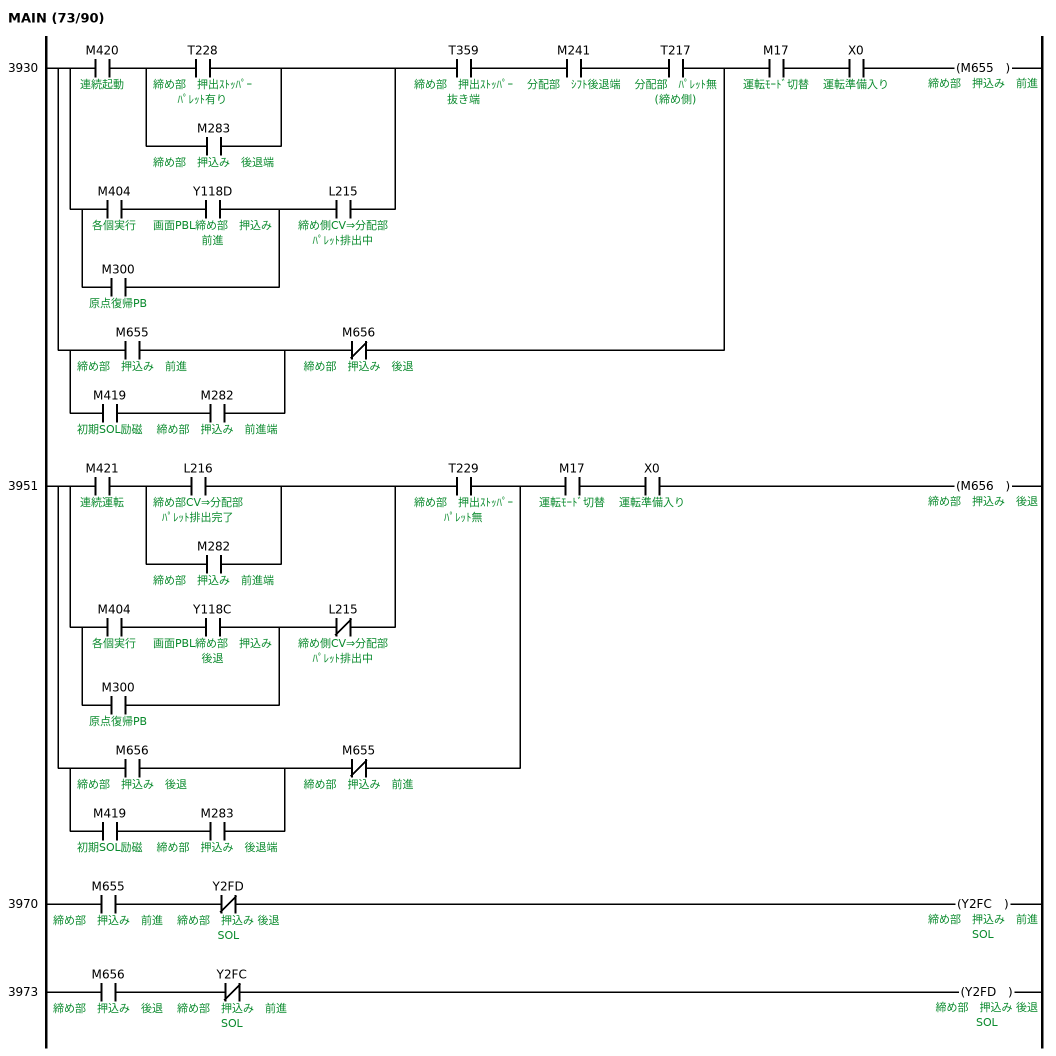
[picture p72: ladder of MAIN, rungs at steps 3930 to 3973]
3930  LD      M420  ; 連続起動
      LD      T228  ; 締め部　押出ｽﾄｯﾊﾟｰ ﾊﾟﾚｯﾄ有り
      OR      M283  ; 締め部　押込み　後退端
      ANB
      LD      M404  ; 各個実行
      AND     Y118D  ; 画面PBL締め部　押込み　前進
      OR      M300  ; 原点復帰PB
      AND     L215  ; 締め側CV⇒分配部 ﾊﾟﾚｯﾄ排出中
      ORB
      AND     T359  ; 締め部　押出ｽﾄｯﾊﾟｰ 抜き端
      AND     M241  ; 分配部　ｼﾌﾄ後退端
      AND     T217  ; 分配部　ﾊﾟﾚｯﾄ無 (締め側)
      LD      M655  ; 締め部　押込み　前進
      LD      M419  ; 初期SOL励磁
      AND     M282  ; 締め部　押込み　前進端
      ORB
      ANI     M656  ; 締め部　押込み　後退
      ORB
      AND     M17  ; 運転ﾓｰﾄﾞ切替
      AND     X0  ; 運転準備入り
      OUT     M655  ; 締め部　押込み　前進
3951  LD      M421  ; 連続運転
      LD      L216  ; 締め部CV⇒分配部 ﾊﾟﾚｯﾄ排出完了
      OR      M282  ; 締め部　押込み　前進端
      ANB
      LD      M404  ; 各個実行
      AND     Y118C  ; 画面PBL締め部　押込み　後退
      OR      M300  ; 原点復帰PB
      ANI     L215  ; 締め側CV⇒分配部 ﾊﾟﾚｯﾄ排出中
      ORB
      AND     T229  ; 締め部　押出ｽﾄｯﾊﾟｰ ﾊﾟﾚｯﾄ無
      LD      M656  ; 締め部　押込み　後退
      LD      M419  ; 初期SOL励磁
      AND     M283  ; 締め部　押込み　後退端
      ORB
      ANI     M655  ; 締め部　押込み　前進
      ORB
      AND     M17  ; 運転ﾓｰﾄﾞ切替
      AND     X0  ; 運転準備入り
      OUT     M656  ; 締め部　押込み　後退
3970  LD      M655  ; 締め部　押込み　前進
      ANI     Y2FD  ; 締め部　押込み 後退 SOL
      OUT     Y2FC  ; 締め部　押込み　前進 SOL
3973  LD      M656  ; 締め部　押込み　後退
      ANI     Y2FC  ; 締め部　押込み　前進 SOL
      OUT     Y2FD  ; 締め部　押込み 後退 SOL
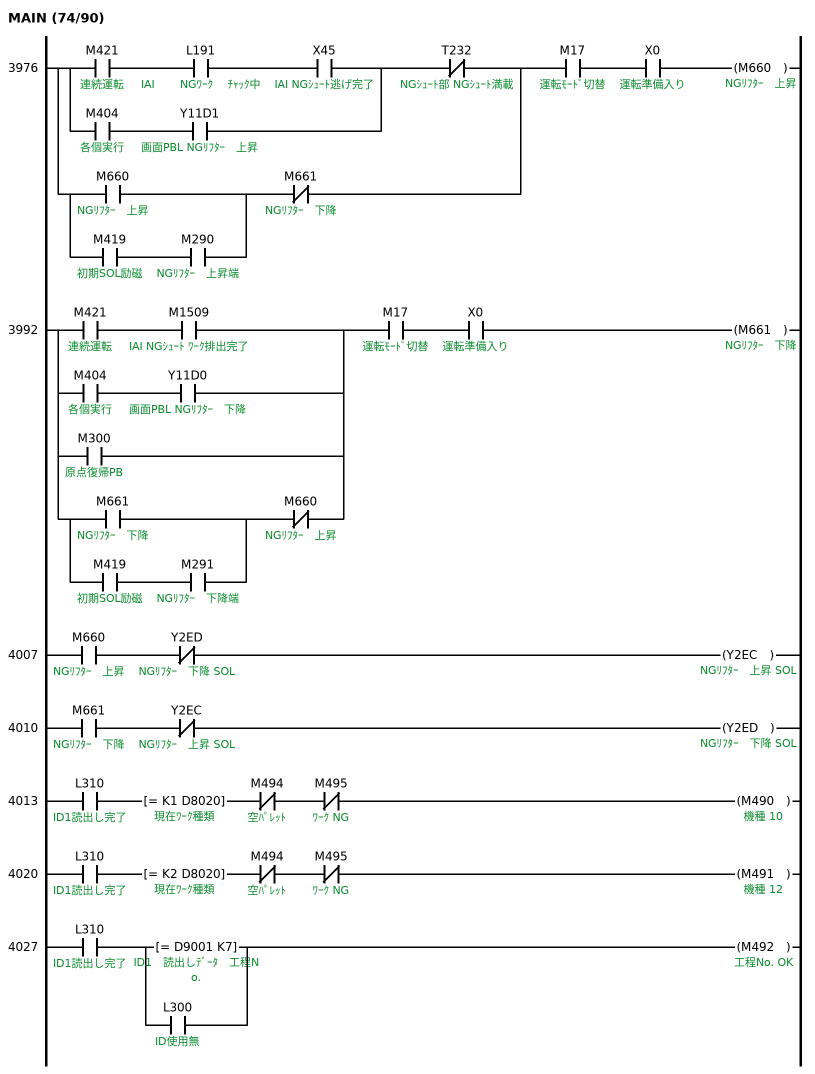
3976  LD      M421  ; 連続運転
      AND     L191  ; IAI　　 NGﾜｰｸ　 ﾁｬｯｸ中
      AND     X45  ; IAI NGｼｭｰﾄ逃げ完了
      LD      M404  ; 各個実行
      AND     Y11D1  ; 画面PBL NGﾘﾌﾀｰ　上昇
      ORB
      ANI     T232  ; NGｼｭｰﾄ部 NGｼｭｰﾄ満載
      LD      M660  ; NGﾘﾌﾀｰ　上昇
      LD      M419  ; 初期SOL励磁
      AND     M290  ; NGﾘﾌﾀｰ　上昇端
      ORB
      ANI     M661  ; NGﾘﾌﾀｰ　下降
      ORB
      AND     M17  ; 運転ﾓｰﾄﾞ切替
      AND     X0  ; 運転準備入り
      OUT     M660  ; NGﾘﾌﾀｰ　上昇
3992  LD      M421  ; 連続運転
      AND     M1509  ; IAI NGｼｭｰﾄ ﾜｰｸ排出完了
      LD      M404  ; 各個実行
      AND     Y11D0  ; 画面PBL NGﾘﾌﾀｰ　下降
      ORB
      OR      M300  ; 原点復帰PB
      LD      M661  ; NGﾘﾌﾀｰ　下降
      LD      M419  ; 初期SOL励磁
      AND     M291  ; NGﾘﾌﾀｰ　下降端
      ORB
      ANI     M660  ; NGﾘﾌﾀｰ　上昇
      ORB
      AND     M17  ; 運転ﾓｰﾄﾞ切替
      AND     X0  ; 運転準備入り
      OUT     M661  ; NGﾘﾌﾀｰ　下降
4007  LD      M660  ; NGﾘﾌﾀｰ　上昇
      ANI     Y2ED  ; NGﾘﾌﾀｰ　下降 SOL
      OUT     Y2EC  ; NGﾘﾌﾀｰ　上昇 SOL
4010  LD      M661  ; NGﾘﾌﾀｰ　下降
      ANI     Y2EC  ; NGﾘﾌﾀｰ　上昇 SOL
      OUT     Y2ED  ; NGﾘﾌﾀｰ　下降 SOL
4013  LD      L310  ; ID1読出し完了
      AND=    K1 D8020  ; 現在ﾜｰｸ種類
      ANI     M494  ; 空ﾊﾟﾚｯﾄ
      ANI     M495  ; ﾜｰｸ NG
      OUT     M490  ; 機種 10
4020  LD      L310  ; ID1読出し完了
      AND=    K2 D8020  ; 現在ﾜｰｸ種類
      ANI     M494  ; 空ﾊﾟﾚｯﾄ
      ANI     M495  ; ﾜｰｸ NG
      OUT     M491  ; 機種 12
4027  LD      L310  ; ID1読出し完了
      LD=     D9001 K7  ; ID1　読出しﾃﾞｰﾀ　工程No.
      OR      L300  ; ID使用無
      ANB
      OUT     M492  ; 工程No. OK
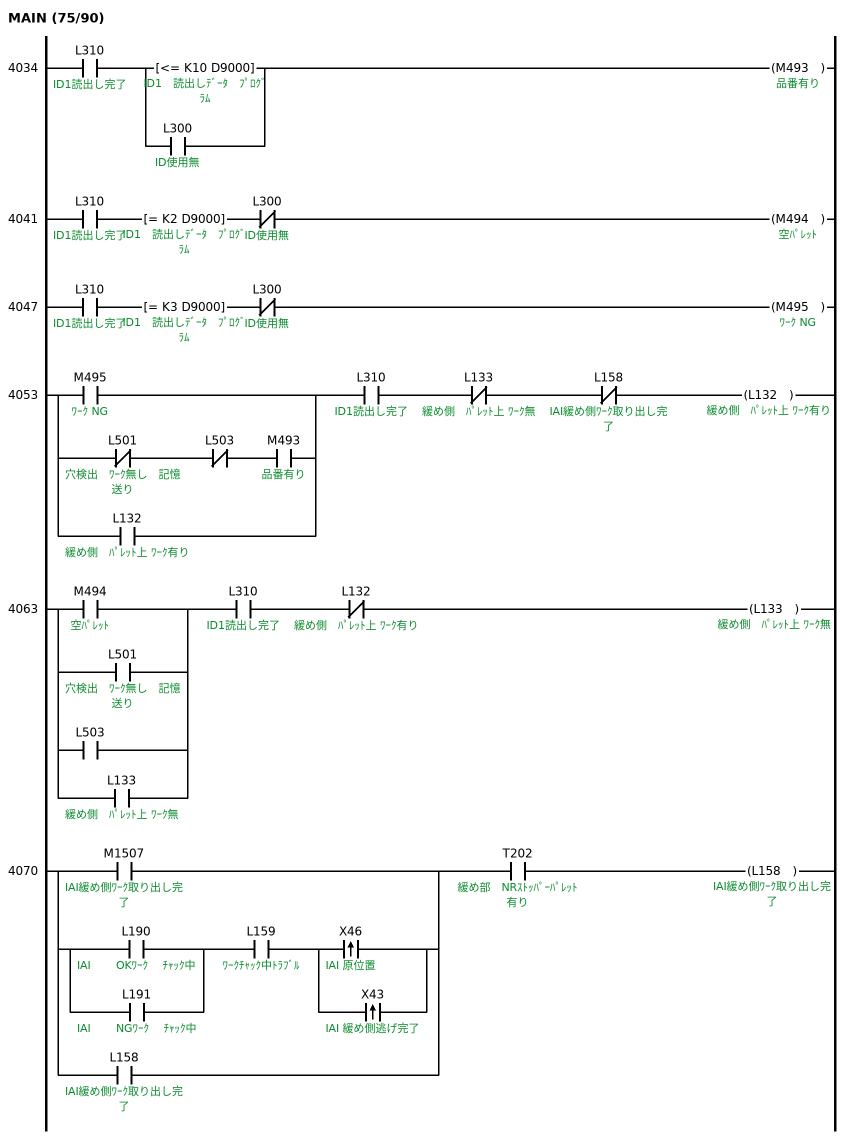
4034  LD      L310  ; ID1読出し完了
      LD<=    K10 D9000  ; ID1　読出しﾃﾞｰﾀ　ﾌﾟﾛｸﾞﾗﾑ
      OR      L300  ; ID使用無
      ANB
      OUT     M493  ; 品番有り
4041  LD      L310  ; ID1読出し完了
      AND=    K2 D9000  ; ID1　読出しﾃﾞｰﾀ　ﾌﾟﾛｸﾞﾗﾑ
      ANI     L300  ; ID使用無
      OUT     M494  ; 空ﾊﾟﾚｯﾄ
4047  LD      L310  ; ID1読出し完了
      AND=    K3 D9000  ; ID1　読出しﾃﾞｰﾀ　ﾌﾟﾛｸﾞﾗﾑ
      ANI     L300  ; ID使用無
      OUT     M495  ; ﾜｰｸ NG
4053  LD      M495  ; ﾜｰｸ NG
      LDI     L501  ; 穴検出　ﾜｰｸ無し　記憶送り
      ANI     L503
      AND     M493  ; 品番有り
      ORB
      OR      L132  ; 緩め側　ﾊﾟﾚｯﾄ上 ﾜｰｸ有り
      AND     L310  ; ID1読出し完了
      ANI     L133  ; 緩め側　ﾊﾟﾚｯﾄ上 ﾜｰｸ無
      ANI     L158  ; IAI緩め側ﾜｰｸ取り出し完了
      OUT     L132  ; 緩め側　ﾊﾟﾚｯﾄ上 ﾜｰｸ有り
4063  LD      M494  ; 空ﾊﾟﾚｯﾄ
      OR      L501  ; 穴検出　ﾜｰｸ無し　記憶送り
      OR      L503
      OR      L133  ; 緩め側　ﾊﾟﾚｯﾄ上 ﾜｰｸ無
      AND     L310  ; ID1読出し完了
      ANI     L132  ; 緩め側　ﾊﾟﾚｯﾄ上 ﾜｰｸ有り
      OUT     L133  ; 緩め側　ﾊﾟﾚｯﾄ上 ﾜｰｸ無
4070  LD      M1507  ; IAI緩め側ﾜｰｸ取り出し完了
      LD      L190  ; IAI　　 OKﾜｰｸ　 ﾁｬｯｸ中
      OR      L191  ; IAI　　 NGﾜｰｸ　 ﾁｬｯｸ中
      AND     L159  ; ﾜｰｸﾁｬｯｸ中ﾄﾗﾌﾞﾙ
      LDP     X46  ; IAI 原位置
      ORP     X43  ; IAI 緩め側逃げ完了
      ANB
      ORB
      OR      L158  ; IAI緩め側ﾜｰｸ取り出し完了
      AND     T202  ; 緩め部　NRｽﾄｯﾊﾟｰﾊﾟﾚｯﾄ有り
      OUT     L158  ; IAI緩め側ﾜｰｸ取り出し完了
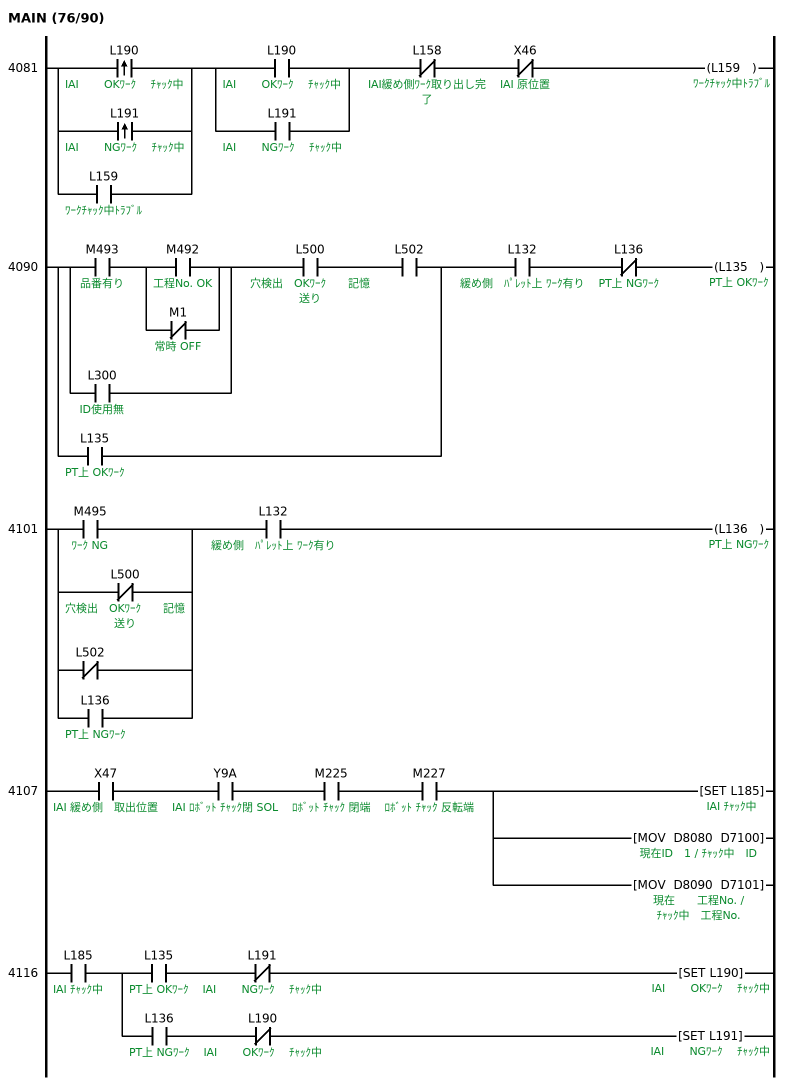
4081  LDP     L190  ; IAI　　 OKﾜｰｸ　 ﾁｬｯｸ中
      ORP     L191  ; IAI　　 NGﾜｰｸ　 ﾁｬｯｸ中
      OR      L159  ; ﾜｰｸﾁｬｯｸ中ﾄﾗﾌﾞﾙ
      LD      L190  ; IAI　　 OKﾜｰｸ　 ﾁｬｯｸ中
      OR      L191  ; IAI　　 NGﾜｰｸ　 ﾁｬｯｸ中
      ANB
      ANI     L158  ; IAI緩め側ﾜｰｸ取り出し完了
      ANI     X46  ; IAI 原位置
      OUT     L159  ; ﾜｰｸﾁｬｯｸ中ﾄﾗﾌﾞﾙ
4090  LD      M493  ; 品番有り
      LD      M492  ; 工程No. OK
      ORI     M1  ; 常時 OFF
      ANB
      OR      L300  ; ID使用無
      AND     L500  ; 穴検出　OKﾜｰｸ　　記憶送り
      AND     L502
      OR      L135  ; PT上 OKﾜｰｸ
      AND     L132  ; 緩め側　ﾊﾟﾚｯﾄ上 ﾜｰｸ有り
      ANI     L136  ; PT上 NGﾜｰｸ
      OUT     L135  ; PT上 OKﾜｰｸ
4101  LD      M495  ; ﾜｰｸ NG
      ORI     L500  ; 穴検出　OKﾜｰｸ　　記憶送り
      ORI     L502
      OR      L136  ; PT上 NGﾜｰｸ
      AND     L132  ; 緩め側　ﾊﾟﾚｯﾄ上 ﾜｰｸ有り
      OUT     L136  ; PT上 NGﾜｰｸ
4107  LD      X47  ; IAI 緩め側　取出位置
      AND     Y9A  ; IAI ﾛﾎﾞｯﾄ ﾁｬｯｸ閉 SOL
      AND     M225  ; ﾛﾎﾞｯﾄ ﾁｬｯｸ 閉端
      AND     M227  ; ﾛﾎﾞｯﾄ ﾁｬｯｸ 反転端
      SET     L185  ; IAI ﾁｬｯｸ中
      MOV     D8080 D7100  ; 現在ID　1 / ﾁｬｯｸ中　ID
      MOV     D8090 D7101  ; 現在　　工程No. / ﾁｬｯｸ中　工程No.
4116  LD      L185  ; IAI ﾁｬｯｸ中
      MPS
      AND     L135  ; PT上 OKﾜｰｸ
      ANI     L191  ; IAI　　 NGﾜｰｸ　 ﾁｬｯｸ中
      SET     L190  ; IAI　　 OKﾜｰｸ　 ﾁｬｯｸ中
      MPP
      AND     L136  ; PT上 NGﾜｰｸ
      ANI     L190  ; IAI　　 OKﾜｰｸ　 ﾁｬｯｸ中
      SET     L191  ; IAI　　 NGﾜｰｸ　 ﾁｬｯｸ中
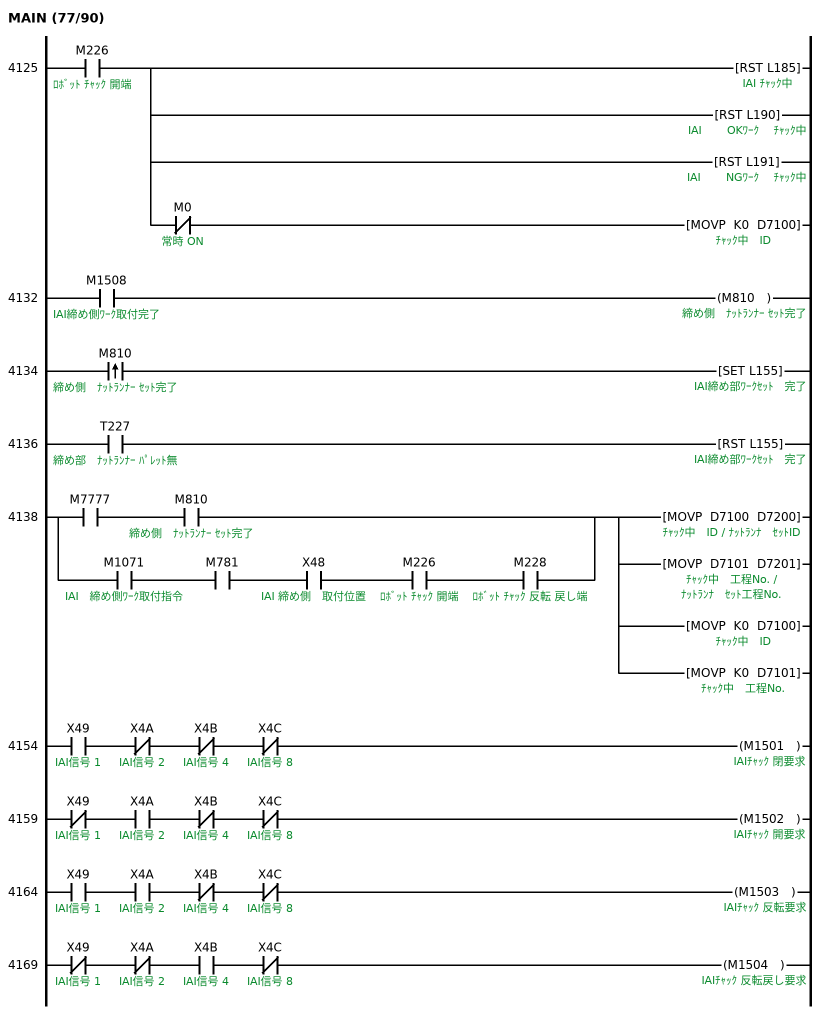
4125  LD      M226  ; ﾛﾎﾞｯﾄ ﾁｬｯｸ 開端
      RST     L185  ; IAI ﾁｬｯｸ中
      RST     L190  ; IAI　　 OKﾜｰｸ　 ﾁｬｯｸ中
      RST     L191  ; IAI　　 NGﾜｰｸ　 ﾁｬｯｸ中
      ANI     M0  ; 常時 ON
      MOVP    K0 D7100
4132  LD      M1508  ; IAI締め側ﾜｰｸ取付完了
      OUT     M810  ; 締め側　ﾅｯﾄﾗﾝﾅｰ ｾｯﾄ完了
4134  LDP     M810  ; 締め側　ﾅｯﾄﾗﾝﾅｰ ｾｯﾄ完了
      SET     L155  ; IAI締め部ﾜｰｸｾｯﾄ　完了
4136  LD      T227  ; 締め部　ﾅｯﾄﾗﾝﾅｰ ﾊﾟﾚｯﾄ無
      RST     L155  ; IAI締め部ﾜｰｸｾｯﾄ　完了
4138  LD      M7777
      AND     M810  ; 締め側　ﾅｯﾄﾗﾝﾅｰ ｾｯﾄ完了
      LD      M1071  ; IAI　締め側ﾜｰｸ取付指令
      AND     M781
      AND     X48  ; IAI 締め側　取付位置
      AND     M226  ; ﾛﾎﾞｯﾄ ﾁｬｯｸ 開端
      AND     M228  ; ﾛﾎﾞｯﾄ ﾁｬｯｸ 反転 戻し端
      ORB
      MOVP    D7100 D7200  ; ﾅｯﾄﾗﾝﾅ　ｾｯﾄID
      MOVP    D7101 D7201  ; ﾅｯﾄﾗﾝﾅ　ｾｯﾄ工程No.
      MOVP    K0 D7100
      MOVP    K0 D7101
4154  LD      X49  ; IAI信号 1
      ANI     X4A  ; IAI信号 2
      ANI     X4B  ; IAI信号 4
      ANI     X4C  ; IAI信号 8
      OUT     M1501  ; IAIﾁｬｯｸ 閉要求
4159  LDI     X49  ; IAI信号 1
      AND     X4A  ; IAI信号 2
      ANI     X4B  ; IAI信号 4
      ANI     X4C  ; IAI信号 8
      OUT     M1502  ; IAIﾁｬｯｸ 開要求
4164  LD      X49  ; IAI信号 1
      AND     X4A  ; IAI信号 2
      ANI     X4B  ; IAI信号 4
      ANI     X4C  ; IAI信号 8
      OUT     M1503  ; IAIﾁｬｯｸ 反転要求
4169  LDI     X49  ; IAI信号 1
      ANI     X4A  ; IAI信号 2
      AND     X4B  ; IAI信号 4
      ANI     X4C  ; IAI信号 8
      OUT     M1504  ; IAIﾁｬｯｸ 反転戻し要求
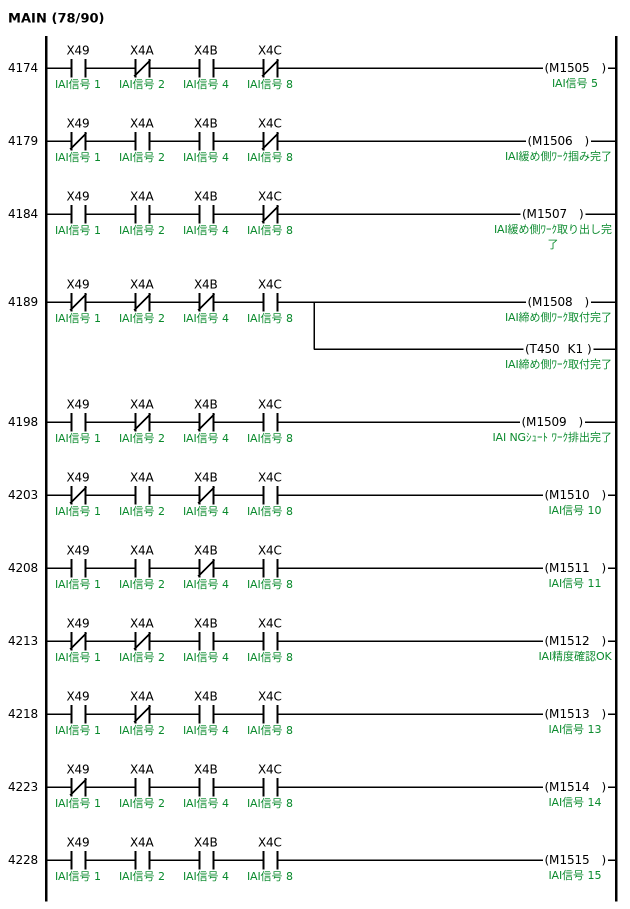
4174  LD      X49  ; IAI信号 1
      ANI     X4A  ; IAI信号 2
      AND     X4B  ; IAI信号 4
      ANI     X4C  ; IAI信号 8
      OUT     M1505  ; IAI信号 5
4179  LDI     X49  ; IAI信号 1
      AND     X4A  ; IAI信号 2
      AND     X4B  ; IAI信号 4
      ANI     X4C  ; IAI信号 8
      OUT     M1506  ; IAI緩め側ﾜｰｸ掴み完了
4184  LD      X49  ; IAI信号 1
      AND     X4A  ; IAI信号 2
      AND     X4B  ; IAI信号 4
      ANI     X4C  ; IAI信号 8
      OUT     M1507  ; IAI緩め側ﾜｰｸ取り出し完了
4189  LDI     X49  ; IAI信号 1
      ANI     X4A  ; IAI信号 2
      ANI     X4B  ; IAI信号 4
      AND     X4C  ; IAI信号 8
      OUT     M1508  ; IAI締め側ﾜｰｸ取付完了
      OUT     T450 K1  ; IAI締め側ﾜｰｸ取付完了
4198  LD      X49  ; IAI信号 1
      ANI     X4A  ; IAI信号 2
      ANI     X4B  ; IAI信号 4
      AND     X4C  ; IAI信号 8
      OUT     M1509  ; IAI NGｼｭｰﾄ ﾜｰｸ排出完了
4203  LDI     X49  ; IAI信号 1
      AND     X4A  ; IAI信号 2
      ANI     X4B  ; IAI信号 4
      AND     X4C  ; IAI信号 8
      OUT     M1510  ; IAI信号 10
4208  LD      X49  ; IAI信号 1
      AND     X4A  ; IAI信号 2
      ANI     X4B  ; IAI信号 4
      AND     X4C  ; IAI信号 8
      OUT     M1511  ; IAI信号 11
4213  LDI     X49  ; IAI信号 1
      ANI     X4A  ; IAI信号 2
      AND     X4B  ; IAI信号 4
      AND     X4C  ; IAI信号 8
      OUT     M1512  ; IAI精度確認OK
4218  LD      X49  ; IAI信号 1
      ANI     X4A  ; IAI信号 2
      AND     X4B  ; IAI信号 4
      AND     X4C  ; IAI信号 8
      OUT     M1513  ; IAI信号 13
4223  LDI     X49  ; IAI信号 1
      AND     X4A  ; IAI信号 2
      AND     X4B  ; IAI信号 4
      AND     X4C  ; IAI信号 8
      OUT     M1514  ; IAI信号 14
4228  LD      X49  ; IAI信号 1
      AND     X4A  ; IAI信号 2
      AND     X4B  ; IAI信号 4
      AND     X4C  ; IAI信号 8
      OUT     M1515  ; IAI信号 15
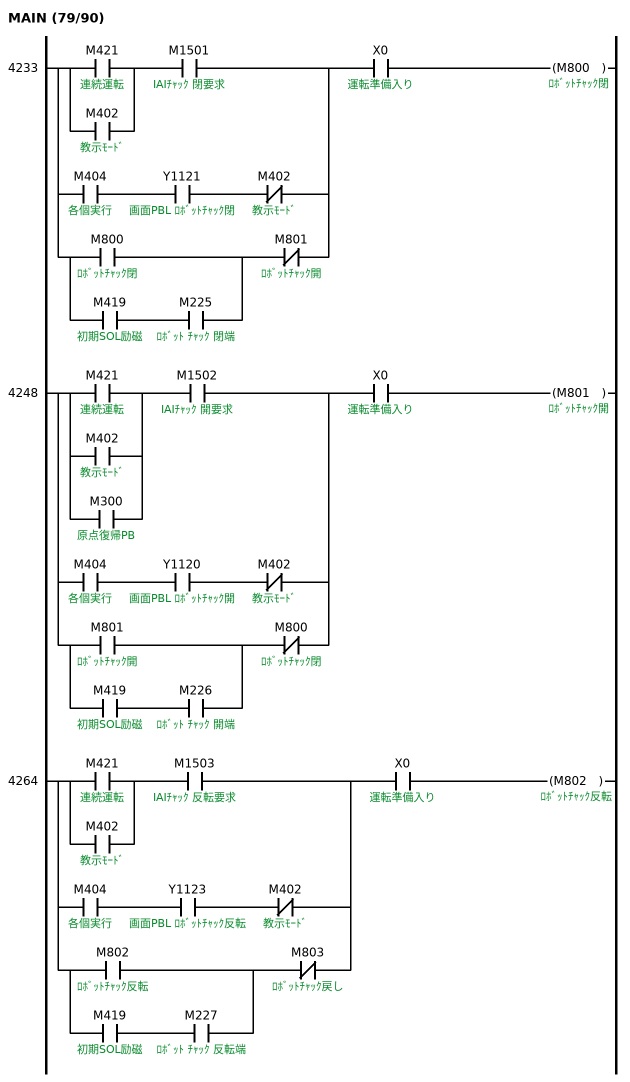
4233  LD      M421  ; 連続運転
      OR      M402  ; 教示ﾓｰﾄﾞ
      AND     M1501  ; IAIﾁｬｯｸ 閉要求
      LD      M404  ; 各個実行
      AND     Y1121  ; 画面PBL ﾛﾎﾞｯﾄﾁｬｯｸ閉
      ANI     M402  ; 教示ﾓｰﾄﾞ
      ORB
      LD      M800  ; ﾛﾎﾞｯﾄﾁｬｯｸ閉
      LD      M419  ; 初期SOL励磁
      AND     M225  ; ﾛﾎﾞｯﾄ ﾁｬｯｸ 閉端
      ORB
      ANI     M801  ; ﾛﾎﾞｯﾄﾁｬｯｸ開
      ORB
      AND     X0  ; 運転準備入り
      OUT     M800  ; ﾛﾎﾞｯﾄﾁｬｯｸ閉
4248  LD      M421  ; 連続運転
      OR      M402  ; 教示ﾓｰﾄﾞ
      OR      M300  ; 原点復帰PB
      AND     M1502  ; IAIﾁｬｯｸ 開要求
      LD      M404  ; 各個実行
      AND     Y1120  ; 画面PBL ﾛﾎﾞｯﾄﾁｬｯｸ開
      ANI     M402  ; 教示ﾓｰﾄﾞ
      ORB
      LD      M801  ; ﾛﾎﾞｯﾄﾁｬｯｸ開
      LD      M419  ; 初期SOL励磁
      AND     M226  ; ﾛﾎﾞｯﾄ ﾁｬｯｸ 開端
      ORB
      ANI     M800  ; ﾛﾎﾞｯﾄﾁｬｯｸ閉
      ORB
      AND     X0  ; 運転準備入り
      OUT     M801  ; ﾛﾎﾞｯﾄﾁｬｯｸ開
4264  LD      M421  ; 連続運転
      OR      M402  ; 教示ﾓｰﾄﾞ
      AND     M1503  ; IAIﾁｬｯｸ 反転要求
      LD      M404  ; 各個実行
      AND     Y1123  ; 画面PBL ﾛﾎﾞｯﾄﾁｬｯｸ反転
      ANI     M402  ; 教示ﾓｰﾄﾞ
      ORB
      LD      M802  ; ﾛﾎﾞｯﾄﾁｬｯｸ反転
      LD      M419  ; 初期SOL励磁
      AND     M227  ; ﾛﾎﾞｯﾄ ﾁｬｯｸ 反転端
      ORB
      ANI     M803  ; ﾛﾎﾞｯﾄﾁｬｯｸ戻し
      ORB
      AND     X0  ; 運転準備入り
      OUT     M802  ; ﾛﾎﾞｯﾄﾁｬｯｸ反転
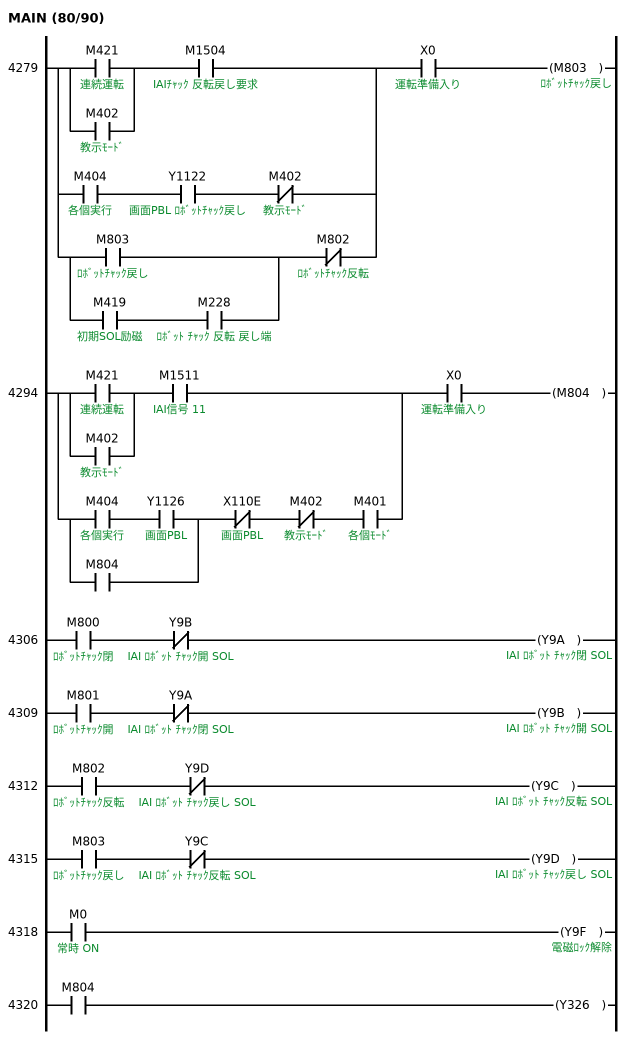
4279  LD      M421  ; 連続運転
      OR      M402  ; 教示ﾓｰﾄﾞ
      AND     M1504  ; IAIﾁｬｯｸ 反転戻し要求
      LD      M404  ; 各個実行
      AND     Y1122  ; 画面PBL ﾛﾎﾞｯﾄﾁｬｯｸ戻し
      ANI     M402  ; 教示ﾓｰﾄﾞ
      ORB
      LD      M803  ; ﾛﾎﾞｯﾄﾁｬｯｸ戻し
      LD      M419  ; 初期SOL励磁
      AND     M228  ; ﾛﾎﾞｯﾄ ﾁｬｯｸ 反転 戻し端
      ORB
      ANI     M802  ; ﾛﾎﾞｯﾄﾁｬｯｸ反転
      ORB
      AND     X0  ; 運転準備入り
      OUT     M803  ; ﾛﾎﾞｯﾄﾁｬｯｸ戻し
4294  LD      M421  ; 連続運転
      OR      M402  ; 教示ﾓｰﾄﾞ
      AND     M1511  ; IAI信号 11
      LD      M404  ; 各個実行
      AND     Y1126  ; 画面PBL
      OR      M804
      ANI     X110E  ; 画面PBL
      ANI     M402  ; 教示ﾓｰﾄﾞ
      AND     M401  ; 各個ﾓｰﾄﾞ
      ORB
      AND     X0  ; 運転準備入り
      OUT     M804
4306  LD      M800  ; ﾛﾎﾞｯﾄﾁｬｯｸ閉
      ANI     Y9B  ; IAI ﾛﾎﾞｯﾄ ﾁｬｯｸ開 SOL
      OUT     Y9A  ; IAI ﾛﾎﾞｯﾄ ﾁｬｯｸ閉 SOL
4309  LD      M801  ; ﾛﾎﾞｯﾄﾁｬｯｸ開
      ANI     Y9A  ; IAI ﾛﾎﾞｯﾄ ﾁｬｯｸ閉 SOL
      OUT     Y9B  ; IAI ﾛﾎﾞｯﾄ ﾁｬｯｸ開 SOL
4312  LD      M802  ; ﾛﾎﾞｯﾄﾁｬｯｸ反転
      ANI     Y9D  ; IAI ﾛﾎﾞｯﾄ ﾁｬｯｸ戻し SOL
      OUT     Y9C  ; IAI ﾛﾎﾞｯﾄ ﾁｬｯｸ反転 SOL
4315  LD      M803  ; ﾛﾎﾞｯﾄﾁｬｯｸ戻し
      ANI     Y9C  ; IAI ﾛﾎﾞｯﾄ ﾁｬｯｸ反転 SOL
      OUT     Y9D  ; IAI ﾛﾎﾞｯﾄ ﾁｬｯｸ戻し SOL
4318  LD      M0  ; 常時 ON
      OUT     Y9F  ; 電磁ﾛｯｸ解除
4320  LD      M804
      OUT     Y326
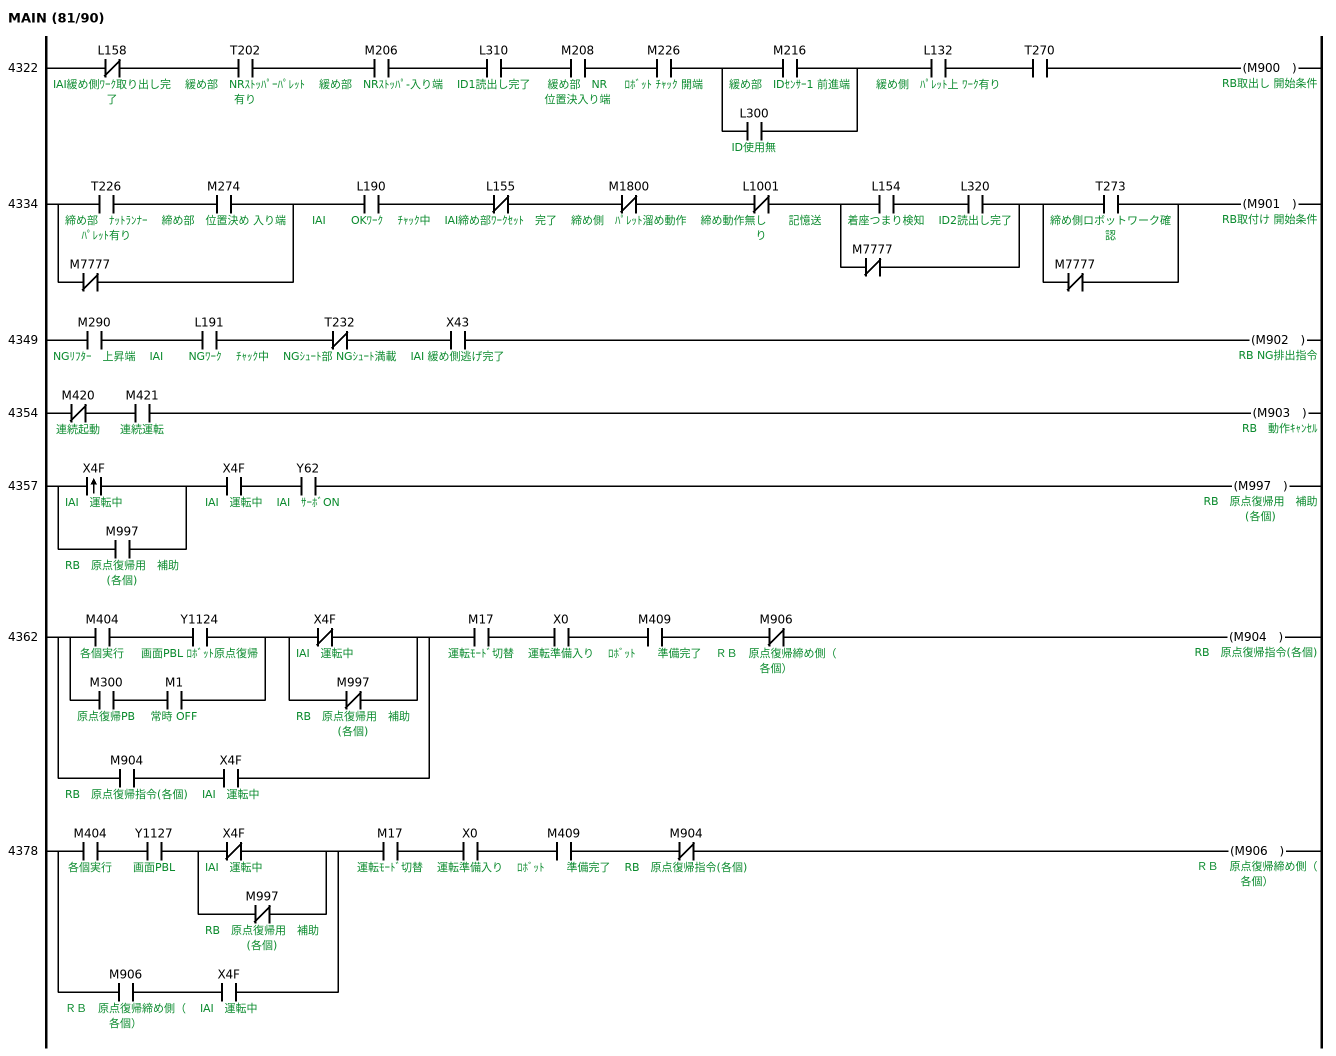
4322  LDI     L158  ; IAI緩め側ﾜｰｸ取り出し完了
      AND     T202  ; 緩め部　NRｽﾄｯﾊﾟｰﾊﾟﾚｯﾄ有り
      AND     M206  ; 緩め部　NRｽﾄｯﾊﾟ-入り端
      AND     L310  ; ID1読出し完了
      AND     M208  ; 緩め部　NR 位置決入り端
      AND     M226  ; ﾛﾎﾞｯﾄ ﾁｬｯｸ 開端
      LD      M216  ; 緩め部　IDｾﾝｻｰ1 前進端
      OR      L300  ; ID使用無
      ANB
      AND     L132  ; 緩め側　ﾊﾟﾚｯﾄ上 ﾜｰｸ有り
      AND     T270
      OUT     M900  ; RB取出し 開始条件
4334  LD      T226  ; 締め部　ﾅｯﾄﾗﾝﾅｰ ﾊﾟﾚｯﾄ有り
      AND     M274  ; 締め部　位置決め 入り端
      ORI     M7777
      AND     L190  ; IAI　　 OKﾜｰｸ　 ﾁｬｯｸ中
      ANI     L155  ; IAI締め部ﾜｰｸｾｯﾄ　完了
      ANI     M1800  ; 締め側　ﾊﾟﾚｯﾄ溜め動作
      ANI     L1001  ; 締め動作無し　　記憶送り
      LD      L154  ; 着座つまり検知
      AND     L320  ; ID2読出し完了
      ORI     M7777
      ANB
      LD      T273  ; 締め側ロボットワーク確認
      ORI     M7777
      ANB
      OUT     M901  ; RB取付け 開始条件
4349  LD      M290  ; NGﾘﾌﾀｰ　上昇端
      AND     L191  ; IAI　　 NGﾜｰｸ　 ﾁｬｯｸ中
      ANI     T232  ; NGｼｭｰﾄ部 NGｼｭｰﾄ満載
      AND     X43  ; IAI 緩め側逃げ完了
      OUT     M902  ; RB NG排出指令
4354  LDI     M420  ; 連続起動
      AND     M421  ; 連続運転
      OUT     M903  ; RB　動作ｷｬﾝｾﾙ
4357  LDP     X4F  ; IAI　運転中
      OR      M997  ; RB　原点復帰用　補助　　 (各個)
      AND     X4F  ; IAI　運転中
      AND     Y62  ; IAI　ｻｰﾎﾞON
      OUT     M997  ; RB　原点復帰用　補助　　 (各個)
4362  LD      M404  ; 各個実行
      AND     Y1124  ; 画面PBL ﾛﾎﾞｯﾄ原点復帰
      LD      M300  ; 原点復帰PB
      AND     M1  ; 常時 OFF
      ORB
      LDI     X4F  ; IAI　運転中
      ORI     M997  ; RB　原点復帰用　補助　　 (各個)
      ANB
      LD      M904  ; RB　原点復帰指令(各個)
      AND     X4F  ; IAI　運転中
      ORB
      AND     M17  ; 運転ﾓｰﾄﾞ切替
      AND     X0  ; 運転準備入り
      AND     M409  ; ﾛﾎﾞｯﾄ　　準備完了
      ANI     M906  ; ＲＢ　原点復帰締め側（各個）
      OUT     M904  ; RB　原点復帰指令(各個)
4378  LD      M404  ; 各個実行
      AND     Y1127  ; 画面PBL
      LDI     X4F  ; IAI　運転中
      ORI     M997  ; RB　原点復帰用　補助　　 (各個)
      ANB
      LD      M906  ; ＲＢ　原点復帰締め側（各個）
      AND     X4F  ; IAI　運転中
      ORB
      AND     M17  ; 運転ﾓｰﾄﾞ切替
      AND     X0  ; 運転準備入り
      AND     M409  ; ﾛﾎﾞｯﾄ　　準備完了
      ANI     M904  ; RB　原点復帰指令(各個)
      OUT     M906  ; ＲＢ　原点復帰締め側（各個）
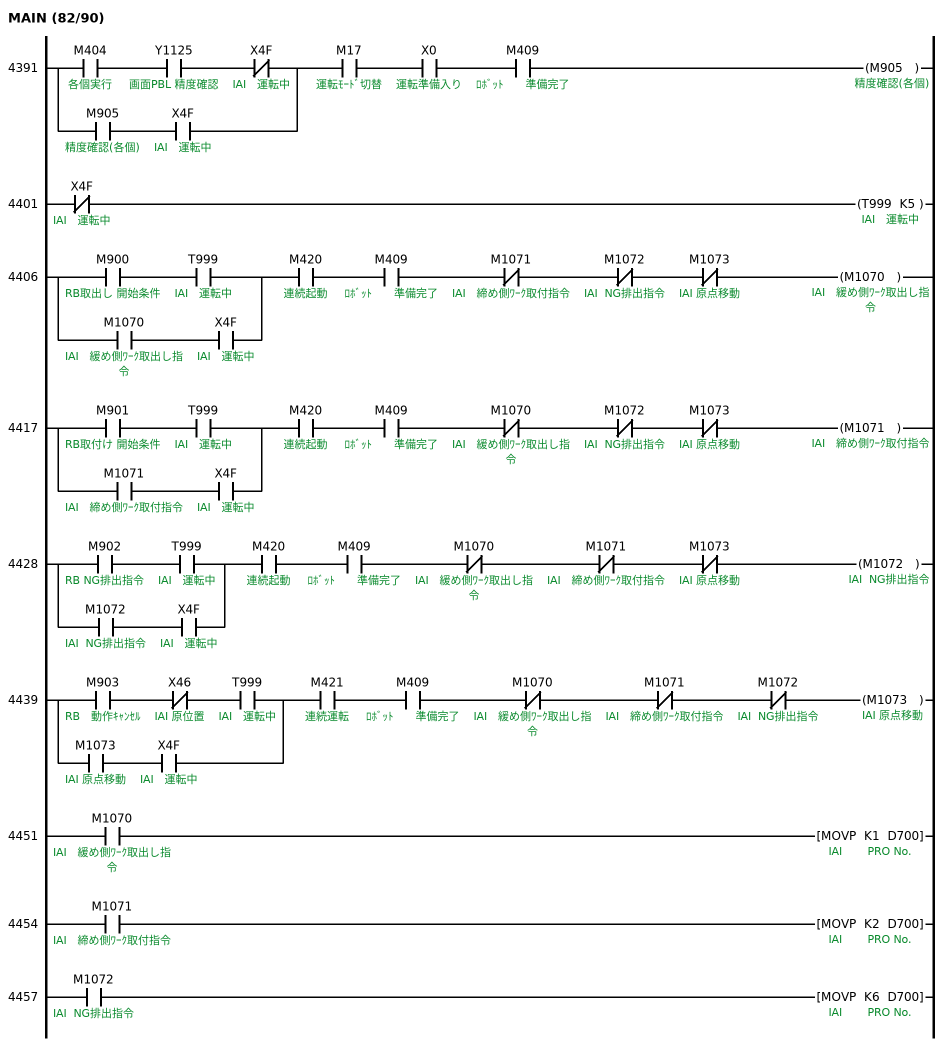
4391  LD      M404  ; 各個実行
      AND     Y1125  ; 画面PBL 精度確認
      ANI     X4F  ; IAI　運転中
      LD      M905  ; 精度確認(各個)
      AND     X4F  ; IAI　運転中
      ORB
      AND     M17  ; 運転ﾓｰﾄﾞ切替
      AND     X0  ; 運転準備入り
      AND     M409  ; ﾛﾎﾞｯﾄ　　準備完了
      OUT     M905  ; 精度確認(各個)
4401  LDI     X4F  ; IAI　運転中
      OUT     T999 K5  ; IAI　運転中
4406  LD      M900  ; RB取出し 開始条件
      AND     T999  ; IAI　運転中
      LD      M1070  ; IAI　緩め側ﾜｰｸ取出し指令
      AND     X4F  ; IAI　運転中
      ORB
      AND     M420  ; 連続起動
      AND     M409  ; ﾛﾎﾞｯﾄ　　準備完了
      ANI     M1071  ; IAI　締め側ﾜｰｸ取付指令
      ANI     M1072  ; IAI  NG排出指令
      ANI     M1073  ; IAI 原点移動
      OUT     M1070  ; IAI　緩め側ﾜｰｸ取出し指令
4417  LD      M901  ; RB取付け 開始条件
      AND     T999  ; IAI　運転中
      LD      M1071  ; IAI　締め側ﾜｰｸ取付指令
      AND     X4F  ; IAI　運転中
      ORB
      AND     M420  ; 連続起動
      AND     M409  ; ﾛﾎﾞｯﾄ　　準備完了
      ANI     M1070  ; IAI　緩め側ﾜｰｸ取出し指令
      ANI     M1072  ; IAI  NG排出指令
      ANI     M1073  ; IAI 原点移動
      OUT     M1071  ; IAI　締め側ﾜｰｸ取付指令
4428  LD      M902  ; RB NG排出指令
      AND     T999  ; IAI　運転中
      LD      M1072  ; IAI  NG排出指令
      AND     X4F  ; IAI　運転中
      ORB
      AND     M420  ; 連続起動
      AND     M409  ; ﾛﾎﾞｯﾄ　　準備完了
      ANI     M1070  ; IAI　緩め側ﾜｰｸ取出し指令
      ANI     M1071  ; IAI　締め側ﾜｰｸ取付指令
      ANI     M1073  ; IAI 原点移動
      OUT     M1072  ; IAI  NG排出指令
4439  LD      M903  ; RB　動作ｷｬﾝｾﾙ
      ANI     X46  ; IAI 原位置
      AND     T999  ; IAI　運転中
      LD      M1073  ; IAI 原点移動
      AND     X4F  ; IAI　運転中
      ORB
      AND     M421  ; 連続運転
      AND     M409  ; ﾛﾎﾞｯﾄ　　準備完了
      ANI     M1070  ; IAI　緩め側ﾜｰｸ取出し指令
      ANI     M1071  ; IAI　締め側ﾜｰｸ取付指令
      ANI     M1072  ; IAI  NG排出指令
      OUT     M1073  ; IAI 原点移動
4451  LD      M1070  ; IAI　緩め側ﾜｰｸ取出し指令
      MOVP    K1 D700  ; IAI　　 PRO No.
4454  LD      M1071  ; IAI　締め側ﾜｰｸ取付指令
      MOVP    K2 D700
4457  LD      M1072  ; IAI  NG排出指令
      MOVP    K6 D700
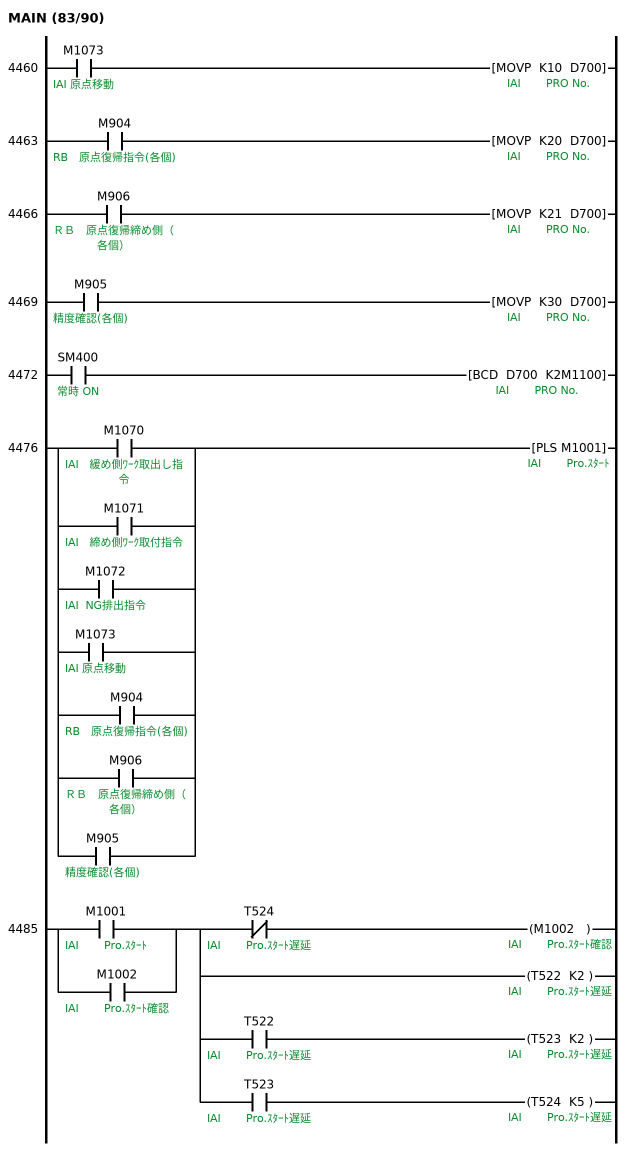
4460  LD      M1073  ; IAI 原点移動
      MOVP    K10 D700
4463  LD      M904  ; RB　原点復帰指令(各個)
      MOVP    K20 D700
4466  LD      M906  ; ＲＢ　原点復帰締め側（各個）
      MOVP    K21 D700
4469  LD      M905  ; 精度確認(各個)
      MOVP    K30 D700
4472  LD      SM400  ; 常時 ON
      BCD     D700 K2M1100  ; RB PRO No.1
4476  LD      M1070  ; IAI　緩め側ﾜｰｸ取出し指令
      OR      M1071  ; IAI　締め側ﾜｰｸ取付指令
      OR      M1072  ; IAI  NG排出指令
      OR      M1073  ; IAI 原点移動
      OR      M904  ; RB　原点復帰指令(各個)
      OR      M906  ; ＲＢ　原点復帰締め側（各個）
      OR      M905  ; 精度確認(各個)
      PLS     M1001  ; IAI　　 Pro.ｽﾀｰﾄ
4485  LD      M1001  ; IAI　　 Pro.ｽﾀｰﾄ
      OR      M1002  ; IAI　　 Pro.ｽﾀｰﾄ確認
      MPS
      ANI     T524  ; IAI　　 Pro.ｽﾀｰﾄ遅延
      OUT     M1002  ; IAI　　 Pro.ｽﾀｰﾄ確認
      MPP
      OUT     T522 K2  ; IAI　　 Pro.ｽﾀｰﾄ遅延
      MPS
      AND     T522  ; IAI　　 Pro.ｽﾀｰﾄ遅延
      OUT     T523 K2  ; IAI　　 Pro.ｽﾀｰﾄ遅延
      MPP
      AND     T523  ; IAI　　 Pro.ｽﾀｰﾄ遅延
      OUT     T524 K5  ; IAI　　 Pro.ｽﾀｰﾄ遅延
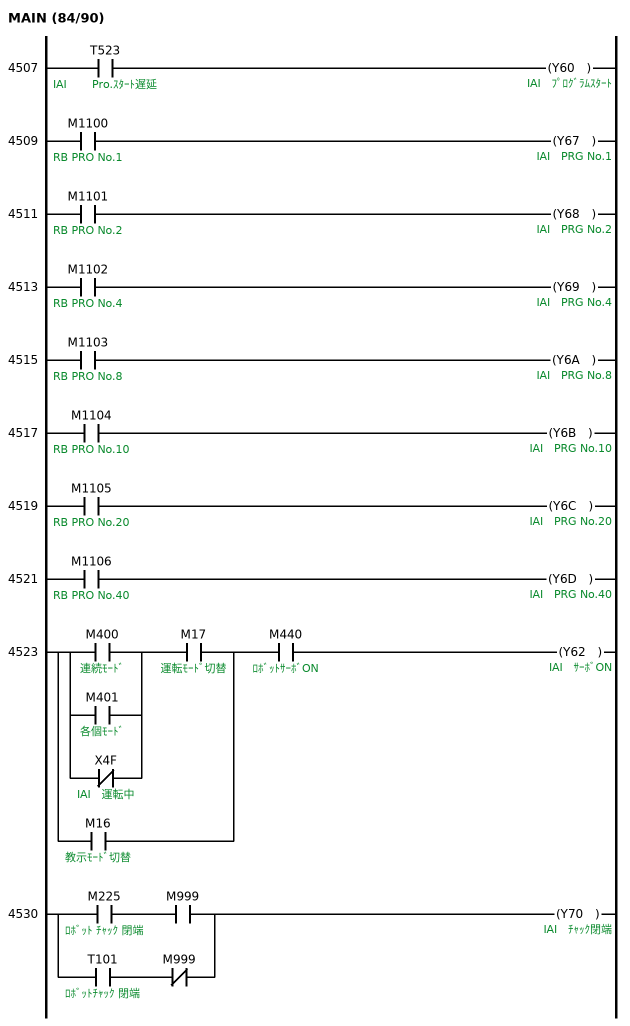
4507  LD      T523  ; IAI　　 Pro.ｽﾀｰﾄ遅延
      OUT     Y60  ; IAI　ﾌﾟﾛｸﾞﾗﾑｽﾀｰﾄ
4509  LD      M1100  ; RB PRO No.1
      OUT     Y67  ; IAI　PRG No.1
4511  LD      M1101  ; RB PRO No.2
      OUT     Y68  ; IAI　PRG No.2
4513  LD      M1102  ; RB PRO No.4
      OUT     Y69  ; IAI　PRG No.4
4515  LD      M1103  ; RB PRO No.8
      OUT     Y6A  ; IAI　PRG No.8
4517  LD      M1104  ; RB PRO No.10
      OUT     Y6B  ; IAI　PRG No.10
4519  LD      M1105  ; RB PRO No.20
      OUT     Y6C  ; IAI　PRG No.20
4521  LD      M1106  ; RB PRO No.40
      OUT     Y6D  ; IAI　PRG No.40
4523  LD      M400  ; 連続ﾓｰﾄﾞ
      OR      M401  ; 各個ﾓｰﾄﾞ
      ORI     X4F  ; IAI　運転中
      AND     M17  ; 運転ﾓｰﾄﾞ切替
      OR      M16  ; 教示ﾓｰﾄﾞ切替
      AND     M440  ; ﾛﾎﾞｯﾄｻｰﾎﾞON
      OUT     Y62  ; IAI　ｻｰﾎﾞON
4530  LD      M225  ; ﾛﾎﾞｯﾄ ﾁｬｯｸ 閉端
      AND     M999
      LD      T101  ; ﾛﾎﾞｯﾄﾁｬｯｸ 閉端
      ANI     M999
      ORB
      OUT     Y70  ; IAI　ﾁｬｯｸ閉端
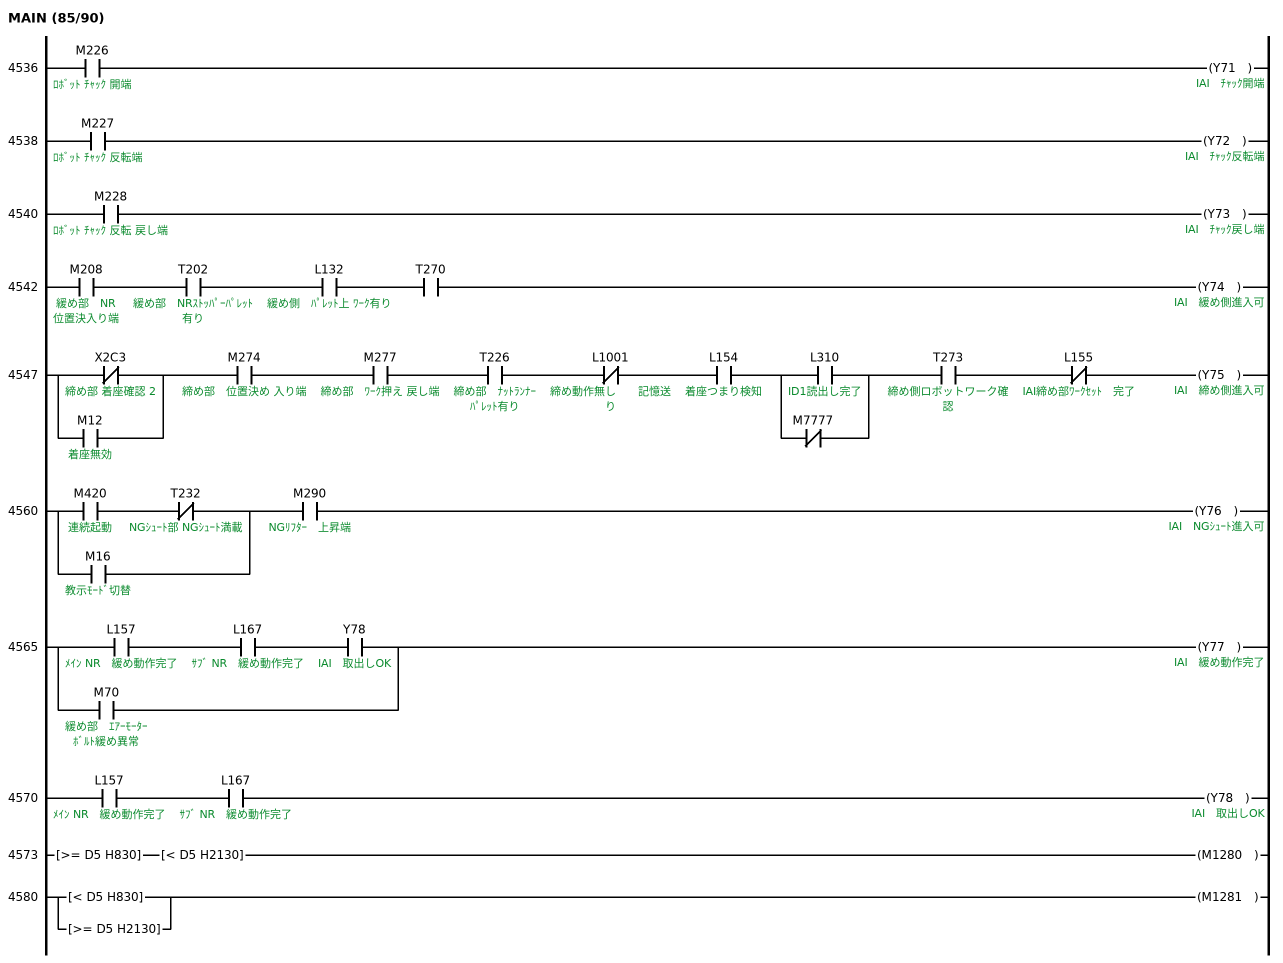
4536  LD      M226  ; ﾛﾎﾞｯﾄ ﾁｬｯｸ 開端
      OUT     Y71  ; IAI　ﾁｬｯｸ開端
4538  LD      M227  ; ﾛﾎﾞｯﾄ ﾁｬｯｸ 反転端
      OUT     Y72  ; IAI　ﾁｬｯｸ反転端
4540  LD      M228  ; ﾛﾎﾞｯﾄ ﾁｬｯｸ 反転 戻し端
      OUT     Y73  ; IAI　ﾁｬｯｸ戻し端
4542  LD      M208  ; 緩め部　NR 位置決入り端
      AND     T202  ; 緩め部　NRｽﾄｯﾊﾟｰﾊﾟﾚｯﾄ有り
      AND     L132  ; 緩め側　ﾊﾟﾚｯﾄ上 ﾜｰｸ有り
      AND     T270
      OUT     Y74  ; IAI　緩め側進入可
4547  LDI     X2C3  ; 締め部 着座確認 2
      OR      M12  ; 着座無効
      AND     M274  ; 締め部　位置決め 入り端
      AND     M277  ; 締め部　ﾜｰｸ押え 戻し端
      AND     T226  ; 締め部　ﾅｯﾄﾗﾝﾅｰ ﾊﾟﾚｯﾄ有り
      ANI     L1001  ; 締め動作無し　　記憶送り
      AND     L154  ; 着座つまり検知
      LD      L310  ; ID1読出し完了
      ORI     M7777
      ANB
      AND     T273  ; 締め側ロボットワーク確認
      ANI     L155  ; IAI締め部ﾜｰｸｾｯﾄ　完了
      OUT     Y75  ; IAI　締め側進入可
4560  LD      M420  ; 連続起動
      ANI     T232  ; NGｼｭｰﾄ部 NGｼｭｰﾄ満載
      OR      M16  ; 教示ﾓｰﾄﾞ切替
      AND     M290  ; NGﾘﾌﾀｰ　上昇端
      OUT     Y76  ; IAI　NGｼｭｰﾄ進入可
4565  LD      L157  ; ﾒｲﾝ NR　緩め動作完了
      AND     L167  ; ｻﾌﾞ NR　緩め動作完了
      AND     Y78  ; IAI　取出しOK
      OR      M70  ; 緩め部　ｴｱｰﾓｰﾀｰ ﾎﾞﾙﾄ緩め異常
      OUT     Y77  ; IAI　緩め動作完了
4570  LD      L157  ; ﾒｲﾝ NR　緩め動作完了
      AND     L167  ; ｻﾌﾞ NR　緩め動作完了
      OUT     Y78  ; IAI　取出しOK
4573  LD>=    D5 H830
      AND<    D5 H2130
      OUT     M1280
4580  LD<     D5 H830
      OR>=    D5 H2130
      OUT     M1281
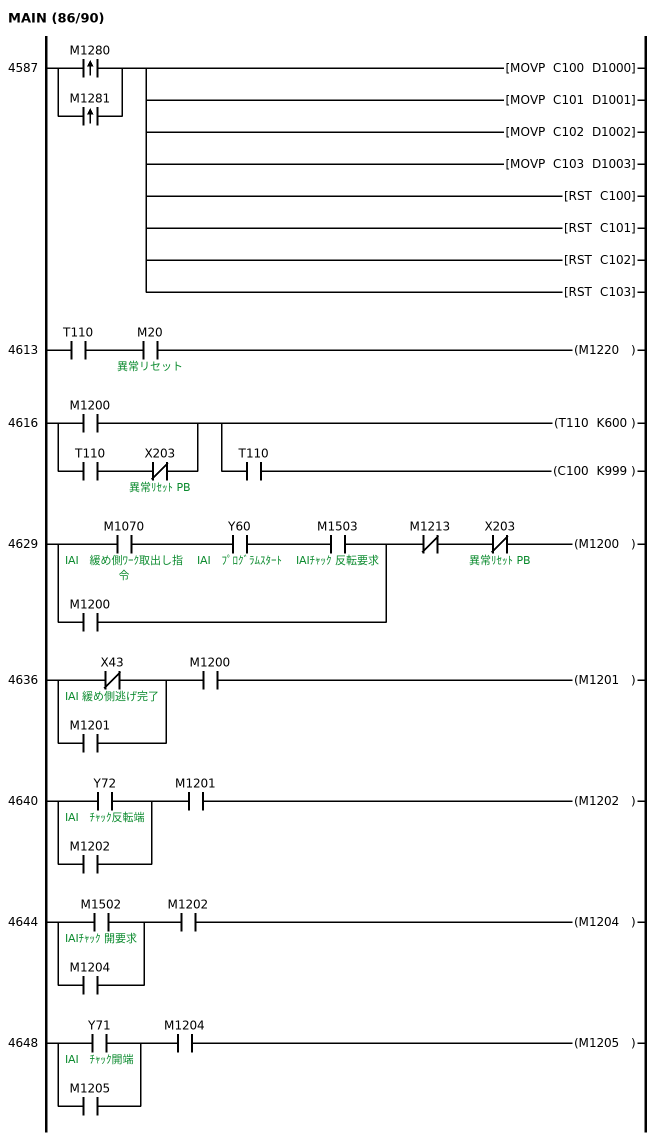
4587  LDP     M1280
      ORP     M1281
      MOVP    C100 D1000
      MOVP    C101 D1001
      MOVP    C102 D1002
      MOVP    C103 D1003
      RST     C100
      RST     C101
      RST     C102
      RST     C103
4613  LD      T110
      AND     M20  ; 異常リセット
      OUT     M1220
4616  LD      M1200
      LD      T110
      ANI     X203  ; 異常ﾘｾｯﾄ PB
      ORB
      OUT     T110 K600
      AND     T110
      OUT     C100 K999
4629  LD      M1070  ; IAI　緩め側ﾜｰｸ取出し指令
      AND     Y60  ; IAI　ﾌﾟﾛｸﾞﾗﾑｽﾀｰﾄ
      AND     M1503  ; IAIﾁｬｯｸ 反転要求
      OR      M1200
      ANI     M1213
      ANI     X203  ; 異常ﾘｾｯﾄ PB
      OUT     M1200
4636  LDI     X43  ; IAI 緩め側逃げ完了
      OR      M1201
      AND     M1200
      OUT     M1201
4640  LD      Y72  ; IAI　ﾁｬｯｸ反転端
      OR      M1202
      AND     M1201
      OUT     M1202
4644  LD      M1502  ; IAIﾁｬｯｸ 開要求
      OR      M1204
      AND     M1202
      OUT     M1204
4648  LD      Y71  ; IAI　ﾁｬｯｸ開端
      OR      M1205
      AND     M1204
      OUT     M1205
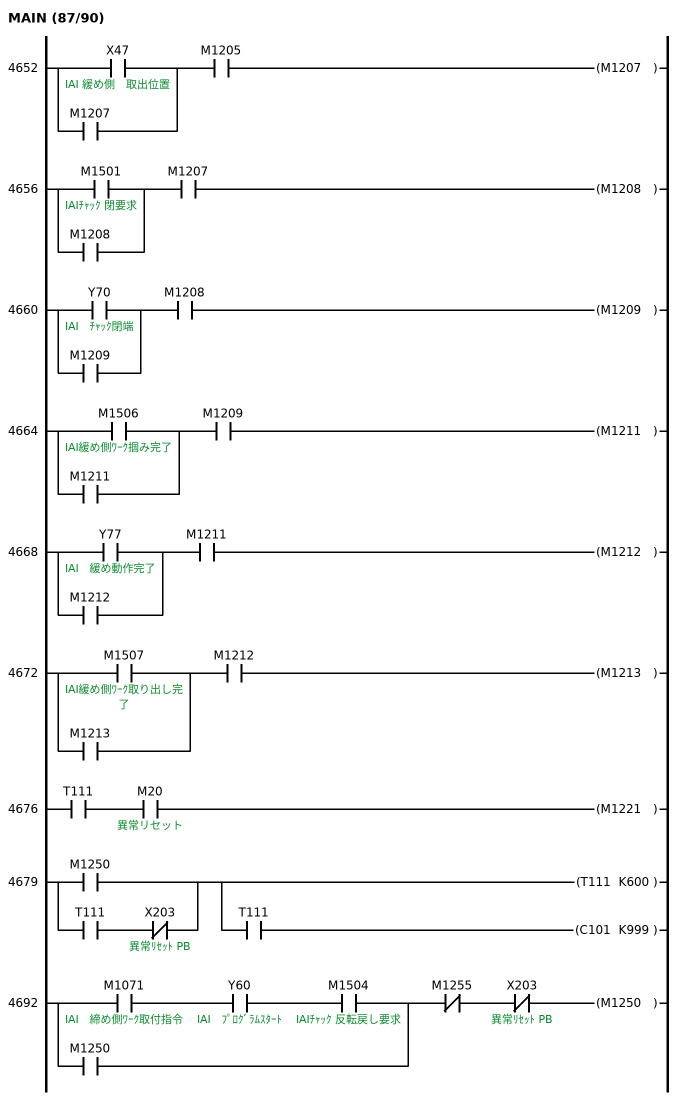
4652  LD      X47  ; IAI 緩め側　取出位置
      OR      M1207
      AND     M1205
      OUT     M1207
4656  LD      M1501  ; IAIﾁｬｯｸ 閉要求
      OR      M1208
      AND     M1207
      OUT     M1208
4660  LD      Y70  ; IAI　ﾁｬｯｸ閉端
      OR      M1209
      AND     M1208
      OUT     M1209
4664  LD      M1506  ; IAI緩め側ﾜｰｸ掴み完了
      OR      M1211
      AND     M1209
      OUT     M1211
4668  LD      Y77  ; IAI　緩め動作完了
      OR      M1212
      AND     M1211
      OUT     M1212
4672  LD      M1507  ; IAI緩め側ﾜｰｸ取り出し完了
      OR      M1213
      AND     M1212
      OUT     M1213
4676  LD      T111
      AND     M20  ; 異常リセット
      OUT     M1221
4679  LD      M1250
      LD      T111
      ANI     X203  ; 異常ﾘｾｯﾄ PB
      ORB
      OUT     T111 K600
      AND     T111
      OUT     C101 K999
4692  LD      M1071  ; IAI　締め側ﾜｰｸ取付指令
      AND     Y60  ; IAI　ﾌﾟﾛｸﾞﾗﾑｽﾀｰﾄ
      AND     M1504  ; IAIﾁｬｯｸ 反転戻し要求
      OR      M1250
      ANI     M1255
      ANI     X203  ; 異常ﾘｾｯﾄ PB
      OUT     M1250
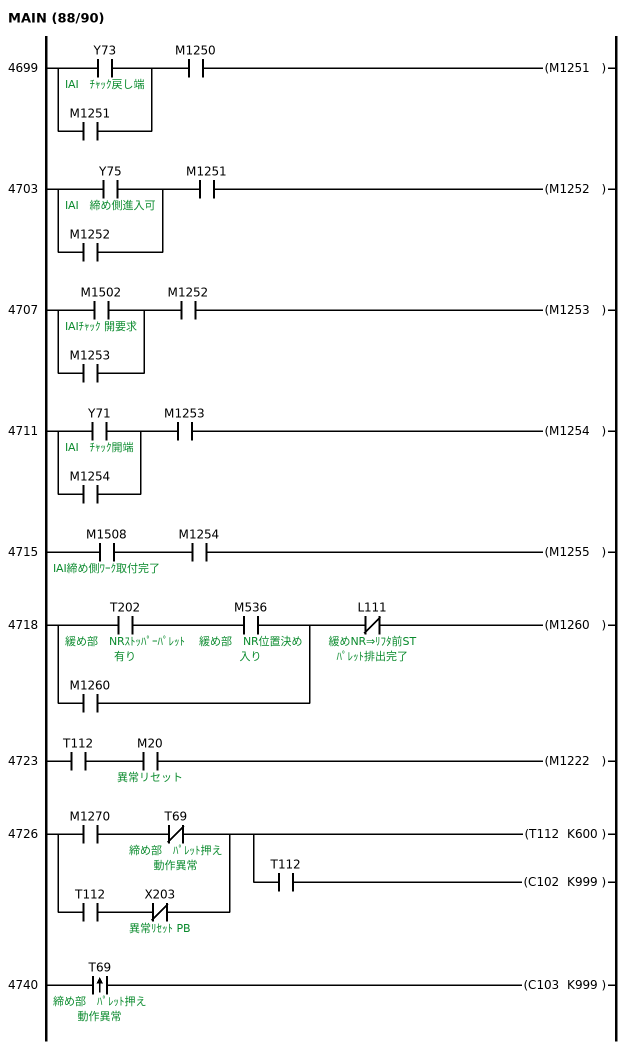
4699  LD      Y73  ; IAI　ﾁｬｯｸ戻し端
      OR      M1251
      AND     M1250
      OUT     M1251
4703  LD      Y75  ; IAI　締め側進入可
      OR      M1252
      AND     M1251
      OUT     M1252
4707  LD      M1502  ; IAIﾁｬｯｸ 開要求
      OR      M1253
      AND     M1252
      OUT     M1253
4711  LD      Y71  ; IAI　ﾁｬｯｸ開端
      OR      M1254
      AND     M1253
      OUT     M1254
4715  LD      M1508  ; IAI締め側ﾜｰｸ取付完了
      AND     M1254
      OUT     M1255
4718  LD      T202  ; 緩め部　NRｽﾄｯﾊﾟｰﾊﾟﾚｯﾄ有り
      AND     M536  ; 緩め部　NR位置決め 入り
      OR      M1260
      ANI     L111  ; 緩めNR⇒ﾘﾌﾀ前ST ﾊﾟﾚｯﾄ排出完了
      OUT     M1260
4723  LD      T112
      AND     M20  ; 異常リセット
      OUT     M1222
4726  LD      M1270
      ANI     T69  ; 締め部　ﾊﾟﾚｯﾄ押え 動作異常
      LD      T112
      ANI     X203  ; 異常ﾘｾｯﾄ PB
      ORB
      OUT     T112 K600
      AND     T112
      OUT     C102 K999
4740  LDP     T69  ; 締め部　ﾊﾟﾚｯﾄ押え 動作異常
      OUT     C103 K999
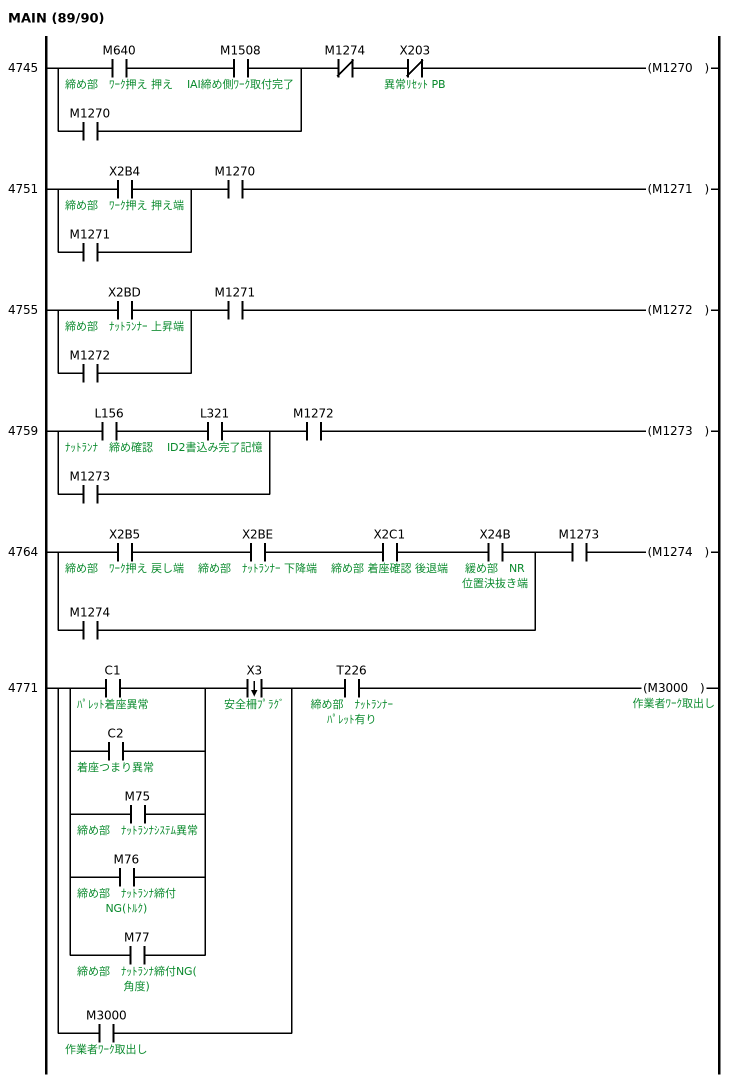
4745  LD      M640  ; 締め部　ﾜｰｸ押え 押え
      AND     M1508  ; IAI締め側ﾜｰｸ取付完了
      OR      M1270
      ANI     M1274
      ANI     X203  ; 異常ﾘｾｯﾄ PB
      OUT     M1270
4751  LD      X2B4  ; 締め部　ﾜｰｸ押え 押え端
      OR      M1271
      AND     M1270
      OUT     M1271
4755  LD      X2BD  ; 締め部　ﾅｯﾄﾗﾝﾅｰ 上昇端
      OR      M1272
      AND     M1271
      OUT     M1272
4759  LD      L156  ; ﾅｯﾄﾗﾝﾅ　締め確認
      AND     L321  ; ID2書込み完了記憶
      OR      M1273
      AND     M1272
      OUT     M1273
4764  LD      X2B5  ; 締め部　ﾜｰｸ押え 戻し端
      AND     X2BE  ; 締め部　ﾅｯﾄﾗﾝﾅｰ 下降端
      AND     X2C1  ; 締め部 着座確認 後退端
      AND     X24B  ; 緩め部　NR 位置決抜き端
      OR      M1274
      AND     M1273
      OUT     M1274
4771  LD      C1  ; ﾊﾟﾚｯﾄ着座異常
      OR      C2  ; 着座つまり異常
      OR      M75  ; 締め部　ﾅｯﾄﾗﾝﾅｼｽﾃﾑ異常
      OR      M76  ; 締め部　ﾅｯﾄﾗﾝﾅ締付 NG(ﾄﾙｸ)
      OR      M77  ; 締め部　ﾅｯﾄﾗﾝﾅ締付NG(角度)
      ANDF    X3  ; 安全柵ﾌﾟﾗｸﾞ
      OR      M3000  ; 作業者ﾜｰｸ取出し
      AND     T226  ; 締め部　ﾅｯﾄﾗﾝﾅｰ ﾊﾟﾚｯﾄ有り
      OUT     M3000  ; 作業者ﾜｰｸ取出し
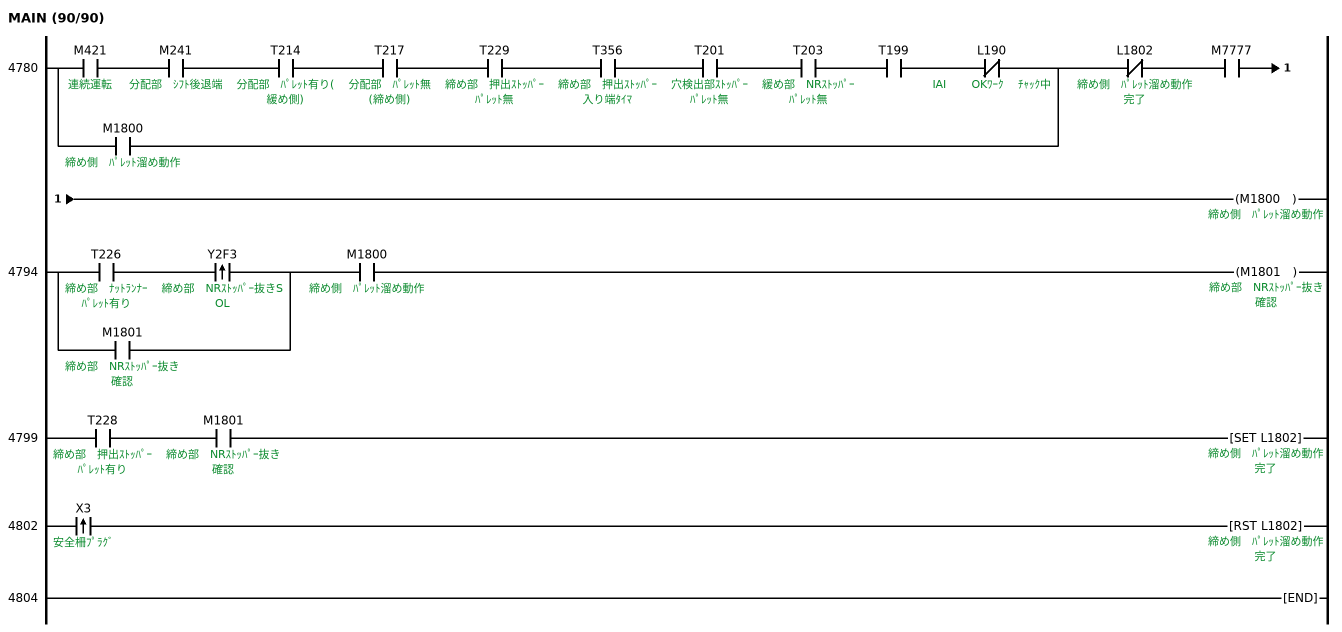
4780  LD      M421  ; 連続運転
      AND     M241  ; 分配部　ｼﾌﾄ後退端
      AND     T214  ; 分配部　ﾊﾟﾚｯﾄ有り(緩め側)
      AND     T217  ; 分配部　ﾊﾟﾚｯﾄ無 (締め側)
      AND     T229  ; 締め部　押出ｽﾄｯﾊﾟｰ ﾊﾟﾚｯﾄ無
      AND     T356  ; 締め部　押出ｽﾄｯﾊﾟｰ 入り端ﾀｲﾏ
      AND     T201  ; 穴検出部ｽﾄｯﾊﾟｰ 　ﾊﾟﾚｯﾄ無
      AND     T203  ; 緩め部　NRｽﾄｯﾊﾟｰ ﾊﾟﾚｯﾄ無
      AND     T199
      ANI     L190  ; IAI　　 OKﾜｰｸ　 ﾁｬｯｸ中
      OR      M1800  ; 締め側　ﾊﾟﾚｯﾄ溜め動作
      ANI     L1802  ; 締め側　ﾊﾟﾚｯﾄ溜め動作完了
      AND     M7777
      OUT     M1800  ; 締め側　ﾊﾟﾚｯﾄ溜め動作
4794  LD      T226  ; 締め部　ﾅｯﾄﾗﾝﾅｰ ﾊﾟﾚｯﾄ有り
      ANDP    Y2F3  ; 締め部　NRｽﾄｯﾊﾟｰ抜きSOL
      OR      M1801  ; 締め部　NRｽﾄｯﾊﾟｰ抜き 確認
      AND     M1800  ; 締め側　ﾊﾟﾚｯﾄ溜め動作
      OUT     M1801  ; 締め部　NRｽﾄｯﾊﾟｰ抜き 確認
4799  LD      T228  ; 締め部　押出ｽﾄｯﾊﾟｰ ﾊﾟﾚｯﾄ有り
      AND     M1801  ; 締め部　NRｽﾄｯﾊﾟｰ抜き 確認
      SET     L1802  ; 締め側　ﾊﾟﾚｯﾄ溜め動作完了
4802  LDP     X3  ; 安全柵ﾌﾟﾗｸﾞ
      RST     L1802  ; 締め側　ﾊﾟﾚｯﾄ溜め動作完了
4804  END
END_PROGRAM

// device comments not shown above
M13  ; 着座有効
M18  ; 払出しON
M21  ; PC電池異常
M22  ; ﾛﾎﾞｯﾄ電池異常
M23  ; ﾌﾟﾗｸﾞ異常
M24  ; ｴｱｰ圧低下
M25  ; CC-LINK異常
M26  ; ﾛﾎﾞｯﾄ異常
M27  ; ﾛﾎﾞｯﾄﾁｬｯｸ LS異常
M28  ; ﾛﾎﾞｯﾄﾁｬｯｸ 反転LS異常
M30  ; 緩め部　押込み　LS異常
M31  ; ｴｱｰﾌﾞﾛｰ ｽﾄｯﾊﾟｰ  LS異常
M32  ; 穴検出部ｽﾄｯﾊﾟｰ　LS異常
M33  ; 緩め部　NRｽﾄｯﾊﾟ-LS異常
M34  ; 緩め部　位置決め LS異常
M36  ; 穴検出部位置決めLS異常
M37  ; 緩め部　ﾅｯﾄﾗﾝﾅ　LS異常
M39  ; 緩め部　ﾘﾌﾀｰ LS異常
M40  ; 緩め部　ﾘﾀｰﾝｴｽｹｰﾌﾟ LS異常
M41  ; 緩め部　ｴｱｰﾌﾞﾛｰ前ｽﾄｯﾊﾟｰ　LS異常
M42  ; 緩め部　穴加工確認LS異常
M43  ; 緩め部　ｼｬｯﾀｰ　　LS異常
M44  ; 緩め部　ﾘﾌﾀｰ前  ｽﾄｯﾊﾟｰ　LS異常
M45  ; 分配部　ｼﾌﾄ LS異常
M46  ; 分配部 着脱ﾌﾟｯｼｬｰ LS異常
M47  ; 緩め部　ﾘﾀｰﾝCV　押出ﾌﾟｯｼｬｰLS異常
M48  ; 緩め部 ﾘﾀｰﾝCV押出前ｽﾄｯﾊﾟｰLS異常
M50  ; 締め部　ﾘﾀｰﾝｴｽｹｰﾌﾟ LS異常
M51  ; 締め部 ﾘﾀｰﾝｽﾄｯﾊﾟｰ LS異常
M53  ; 予備
M54  ; 締め部　ﾘﾌﾀｰ LS異常
M55  ; 締め部　ﾘﾌﾀｰ後　ｽﾄｯﾊﾟｰ　LS異常
M56  ; 締め部　NRｽﾄｯﾊﾟｰLS異常
M57  ; 締め部　位置決め LS異常
M58  ; 締め部 ﾊﾟﾚｯﾄ押え LS異常
M60  ; 締め部　押出ｽﾄｯﾊﾟｰ LS異常
M61  ; 締め部　押込み　LS異常
M62  ; 締め部 ﾅｯﾄﾗﾝﾅｰ　LS異常
M63  ; 締め部　着座確認LS異常
M64  ; NGﾘﾌﾀｰ　LS異常
M65  ; 締め部　IDｾﾝｻｰ　LS異常
M68  ; 穴検出　NG
M69  ; 穴検出　治具折れ異常
M91  ; ID1 異常
M92  ; ID2 異常
M94  ; ﾊﾟﾚｯﾄID異常
M95  ; ID1読み出し異常
M97  ; ID2読み出し異常
M99  ; ID異常
M185  ; ﾅｯﾄﾗﾝﾅTQ HI(ﾄﾙｸ上限NG)
M186  ; ﾅｯﾄﾗﾝﾅTQ LO(ﾄﾙｸ下限NG)
M187  ; ﾅｯﾄﾗﾝﾅBYPASS(軸切)
M190  ; ﾅｯﾄﾗﾝﾅANG HI(角度上限NG)
M191  ; ﾅｯﾄﾗﾝﾅANG LO(角度下限NG)
M288  ; 締め部　IDｾﾝｻｰ2 前進端
M289  ; 締め部　IDｾﾝｻｰ2 後退端
M351  ; 分配部　原位置
M635  ; 締め部　IDｾﾝｻｰ　前進
M636  ; 締め部　IDｾﾝｻｰ　後退
M1107  ; RB PRO No.80
M1600  ; IAI精度確認OK　　確認
M1601  ; IAI精度確認OK　　切り
M2000  ; 品番設定画面
M2001  ; 品番設定可
M2002  ; 設定品番書込み
M2050  ; 品番検索
M2100  ; ワークカウント
M2101  ; カウント一致あり
M2102  ; 新規カウント
M2457  ; ID1 　　読込条件
M2458  ; ID1 　　読込ｽﾀｰﾄ
M2459  ; ID1 　　読込完了
M2470  ; ID2 　　読込条件
M2471  ; ID2 　　読込ｽﾀｰﾄ
M2472  ; ID2 　　読込完了
M2500  ; ID1条件
M2501  ; ID1　 　読出し
M2502  ; ID1　 　TRG ON
M2503  ; ID1　 　TRG OFF
M2504  ; ID1 読出し完了
M2505  ; ID1　読出し異常
M2509  ; ID1　　　書込み　正常終了
M2510  ; ID1　　　書込み
M2511  ; ID1　 　TRG ON
M2512  ; ID1　 　TRG OFF
M2513  ; ID1 書込み完了
M2514  ; ID1　　　書込み　TRG
M2519  ; ID1 TRG ON確認
M2520  ; ID2条件
M2521  ; ID2　 　読出し
M2522  ; ID2　 　TRG ON
M2523  ; ID2　 　TRG OFF
M2524  ; ID2 読出し完了
M2525  ; ID2　読出し異常
M2527  ; ID2　 　読出し　TRG
M2530  ; ID2　　　書込み
M2531  ; ID2　 　TRG ON
M2532  ; ID2　 　TRG OFF
M2533  ; ID2 書込み完了
M2534  ; ID2　　　書込み　TRG
M2539  ; ID2 TRG ON確認
L301  ; 工程番号有り
X1  ; ヒューズ正常
X2  ; エアー元圧正常
X5  ; 緩め側搬送CV INV異常
X6  ; 緩め側ﾘﾌﾄﾓｰﾀｰ ｻｰﾏﾙﾄﾘｯﾌﾟ
X7  ; 緩め側ﾘﾀｰﾝCV INV異常
X8  ; 締め側搬送CV INV異常
X9  ; 締め側ﾘﾌﾄﾓｰﾀｰ ｻｰﾏﾙﾄﾘｯﾌﾟ
X0A  ; 締め側ﾘﾀｰﾝCV INV異常
X0D  ; 着座無効
X0E  ; 電磁ﾛｯｸ 閉
X0F  ; 穴検出部ﾜｰｸ有り
X10  ; 締め部NR OUTDATA 0
X11  ; 締め部NR OUTDATA 1
X12  ; 締め部NR OUTDATA 2
X13  ; 締め部NR OUTDATA 3
X14  ; 締め部NR OUTDATA 4
X15  ; 締め部NR OUTDATA 5
X16  ; 締め部NR OUTDATA 6
X17  ; 締め部NR OUTDATA 7
X37  ; 第1搬送⇒M/C IL　予備
X39  ; 第2ﾊﾟﾚﾘﾀｰﾝC/V IL　干渉外
X3A  ; 第2ﾊﾟﾚﾘﾀｰﾝC/V IL　予備
X3B  ; 第2ﾊﾟﾚﾘﾀｰﾝC/V IL　予備
X40  ; IAI　ｱﾗｰﾑ出力
X42  ; IAI　非常停止出力
X4D  ; IAI ｼｽﾃﾑ ﾒﾓﾘｰ ﾊﾞｯﾃﾘｰ警告
X4E  ; IAI ｱﾌﾞｿﾘｭｰﾄｴﾝｺｰﾀﾞ ﾊﾞｯﾃﾘｰ警告
X50  ; ﾛﾎﾞｯﾄ ﾁｬｯｸ 閉端
X51  ; ﾛﾎﾞｯﾄ ﾁｬｯｸ 開端
X52  ; ﾛﾎﾞｯﾄ ﾁｬｯｸ 反転端
X53  ; ﾛﾎﾞｯﾄ ﾁｬｯｸ 反転 戻し端
X100  ; ID1　　 READ DATA OD0
X101  ; ID1　READ DATA OD1
X102  ; ID1　READ DATA OD2
X103  ; ID1　READ DATA OD3
X104  ; ID1　　 READ DATA OD4
X105  ; ID1　READ DATA OD5
X106  ; ID1　READ DATA OD6
X107  ; ID1　READ DATA OD7
X108  ; ID1　　 NORMAL
X109  ; ID1　　 ERROR
X110  ; ID2　READ DATA OD0
X111  ; ID2　READ DATA OD1
X112  ; ID2　READ DATA OD2
X113  ; ID2　READ DATA OD3
X114  ; ID2　READ DATA OD4
X115  ; ID2　READ DATA OD5
X116  ; ID2　READ DATA OD6
X117  ; ID2　READ DATA OD7
X118  ; ID2　　 NORMAL
X119  ; ID2　　 ERROR
X204  ; 教示 入り SS
X240  ; 緩め部　押込み　前進端
X241  ; 緩め部　押込み　後退端
X243  ; ｴｱｰﾌﾞﾛｰ ｽﾄｯﾊﾟｰ  入り端
X244  ; ｴｱｰﾌﾞﾛｰ ｽﾄｯﾊﾟｰ  抜き端
X245  ; 穴検出部ｽﾄｯﾊﾟｰ　抜き端
X246  ; 穴検出部ｽﾄｯﾊﾟｰ　入り端
X247  ; 緩め部　NRｽﾄｯﾊﾟ-入り端
X248  ; 緩め部　NRｽﾄｯﾊﾟ-抜き端
X24A  ; 緩め部　NR 位置決入り端
X24D  ; NGｼｭｰﾄ部 NGｼｭｰﾄ満載
X24E  ; 穴検出部位置決め入り端
X24F  ; 穴検出部位置決め抜き端
X250  ; 緩め部　ﾒｲﾝ NR  上昇端
X251  ; 緩め部　ﾒｲﾝ NR  下降端
X252  ; 緩め部　IDｾﾝｻｰ　前進端
X253  ; 緩め部　IDｾﾝｻｰ　後退端
X255  ; 緩め部　ﾘﾌﾀｰ上昇端
X256  ; 緩め部　ﾘﾌﾀｰ 下降端
X258  ; 緩め部  穴検出　下降端
X259  ; 緩め部  穴検出　上昇端
X25A  ; 緩め部  穴検出　ｾﾝｻｰ 1
X25B  ; 緩め部  穴検出　ｾﾝｻｰ 2
X25C  ; 緩め部  穴検出　ｾﾝｻｰ 3
X25D  ; 緩め部  穴検出　ｾﾝｻｰ 4
X25E  ; 緩め部　ｻﾌﾞ NR  上昇端
X25F  ; 緩め部　ｻﾌﾞ NR  下降端
X262  ; 緩め部　ﾘﾀｰﾝｴｽｹｰﾌﾟ 前進端
X263  ; 緩め部　ﾘﾀｰﾝｴｽｹｰﾌﾟ 後退端
X264  ; 緩め部　ｴｱｰﾌﾞﾛｰ前ｽﾄｯﾊﾟｰ　入り端
X265  ; 緩め部　ｴｱｰﾌﾞﾛｰ前ｽﾄｯﾊﾟｰ　抜き端
X267  ; 緩め部 ﾘﾀｰﾝCV押出前ｽﾄｯﾊﾟｰ入り端
X268  ; 緩め部 ﾘﾀｰﾝCV押出前ｽﾄｯﾊﾟｰ抜き端
X269  ; 分配部 着脱ﾌﾟｯｼｬ- 前進端
X26A  ; 分配部 着脱ﾌﾟｯｼｬｰ 後退端
X26B  ; 緩め部　ﾘﾌﾀｰ前  ｽﾄｯﾊﾟｰ　入り端
X26C  ; 緩め部　ﾘﾌﾀｰ前  ｽﾄｯﾊﾟｰ　抜き端
X26E  ; 緩め部　ｼｬｯﾀｰ　　開端
X26F  ; 緩め部　ｼｬｯﾀｰ　　閉端
X2A2  ; 締め部　ﾘﾀｰﾝｴｽｹｰﾌﾟ 前進端
X2A3  ; 締め部　ﾘﾀｰﾝｴｽｹｰﾌﾟ 後退端
X2A4  ; 締め部　ﾘﾀｰﾝｽﾄｯﾊﾟｰ 入り端
X2A5  ; 締め部　ﾘﾀｰﾝｽﾄｯﾊﾟｰ 抜き端
X2A7  ; 分配部　ｼﾌﾄ 前進端
X2A8  ; 分配部　ｼﾌﾄ 後退端
X2AB  ; 締め部　ﾘﾌﾀｰ 　　上昇端
X2AC  ; 締め部　ﾘﾌﾀｰ 　　下降端
X2AE  ; 締め部　ﾘﾌﾀｰ後　ｽﾄｯﾊﾟｰ　前進端
X2AF  ; 締め部　ﾘﾌﾀｰ後　ｽﾄｯﾊﾟｰ　後退端
X2B0  ; 締め部　NRｽﾄｯﾊﾟｰ抜き端
X2B1  ; 締め部　NRｽﾄｯﾊﾟｰ入り端
X2B2  ; 締め部　位置決め 入り端
X2B3  ; 締め部　位置決め 抜き端
X2B9  ; 締め部　押出ｽﾄｯﾊﾟｰ 入り端
X2BA  ; 締め部　押出ｽﾄｯﾊﾟｰ 抜き端
X2BB  ; 締め部　押込み　前進端
X2BC  ; 締め部　押込み　後退端
X2C0  ; 締め部 着座確認 前進端
X2C2  ; 締め部　着座確認 1
X2C4  ; 締め部　IDｾﾝｻｰ　前進端
X2C5  ; 締め部　IDｾﾝｻｰ　後退端
X2C6  ; 緩め部　ﾘﾀｰﾝCV　押出ﾘﾌﾀｰ上昇端
X2C7  ; 緩め部　ﾘﾀｰﾝCV　押出ﾘﾌﾀｰ下降端
X2C8  ; NGﾘﾌﾀｰ　上昇端
X2C9  ; NGﾘﾌﾀｰ　下降端
X2CE  ; 緩め部　ﾘﾀｰﾝCV　押出ﾌﾟｯｼｬｰ前進端
X2CF  ; 緩め部　ﾘﾀｰﾝCV　押出ﾌﾟｯｼｬｰ後退端
X1000  ; カウンタオールリセット
X1004  ; ID使用有 PB
X1005  ; ID使用無 PB
X1006  ; 工程No.有 PB
X1007  ; 工程No.無 PB
X1011  ; 品番設定SW
X1050  ; カウントリセット1
X1051  ; カウントリセット2
X1052  ; カウントリセット3
X1053  ; カウントリセット4
X1054  ; カウントリセット5
X1055  ; カウントリセット6
X1056  ; カウントリセット7
X1057  ; カウントリセット8
X1058  ; カウントリセット9
X1059  ; カウントリセット10
X105A  ; カウントリセット11
X1200  ; 設定品番書込み
Y0C9  ; M/C⇒搬送IL ID情報 BCD02
Y0CA  ; M/C⇒搬送IL ID情報 BCD04
Y0CB  ; M/C⇒搬送IL ID情報 BCD08
Y0CC  ; M/C⇒搬送IL ID情報 BCD10
Y0CD  ; M/C⇒搬送IL ID情報 BCD20
Y0CE  ; M/C⇒搬送IL ID情報 BCD40
Y0CF  ; M/C⇒搬送IL ID情報 BCD80
Y120  ; ID1　　 WRITE DATA ID0
Y121  ; ID1　WRITE DATA ID1
Y122  ; ID1　WRITE DATA ID2
Y123  ; ID1　WRITE DATA ID3
Y124  ; ID1　WRITE DATA ID4
Y125  ; ID1　WRITE DATA ID5
Y126  ; ID1　WRITE DATA ID6
Y127  ; ID1　WRITE DATA ID7
Y128  ; ID1　　　R/W
Y129  ; ID1　INHIBIT/TRG
Y130  ; ID2　INHIBIT/TRG
Y131  ; ID2　WRITE DATA ID0
Y132  ; ID2　WRITE DATA ID1
Y133  ; ID2　WRITE DATA ID2
Y134  ; ID2　WRITE DATA ID3
Y135  ; ID2　WRITE DATA ID4
Y136  ; ID2　WRITE DATA ID5
Y137  ; ID2　WRITE DATA ID6
Y138  ; ID2　WRITE DATA ID7
Y139  ; ID2　R/W
Y29E  ; 緩め部　ｼｬｯﾀｰ　　開 SOL
Y29F  ; 緩め部　ｼｬｯﾀｰ　　閉 SOL
Y2EE  ; 締め部　IDｾﾝｻｰ2 前進SOL
Y2EF  ; 締め部　IDｾﾝｻｰ2 後退SOL
Y1004  ; ID使用有 PL
Y1005  ; ID使用無 PL
Y1006  ; 工程番号使用 PL
Y1007  ; 工程番号無し
Y11E6  ; 画面PBL締め部　IDｾﾝｻｰ　後退
Y11E7  ; 画面PBL締め部　IDｾﾝｻｰ　前進
Y1200  ; 設定品番書込み PL
Y1201  ; 機種M10 PBL
Y1202  ; 機種M12 PBL
Y1400  ; 分配部　原位置
Y1401  ; ﾛﾎﾞｯﾄ部　原位置
Y1402  ; 緩め部　原位置
Y1403  ; 締め部　原位置
Y1404  ; NGﾘﾌﾀｰ部原位置
Y1410  ; 分配部ｼﾌﾄ 後退端PL
Y1411  ; 分配部　ｼﾌﾄ 前進端PL
Y1412  ; 分配部 着脱ﾌﾟｯｼｬｰ 後退端PL
Y1413  ; 分配部 着脱ﾌﾟｯｼｬ- 前進端PL
Y1420  ; ﾛﾎﾞｯﾄ ﾁｬｯｸ 開端PL
Y1421  ; ﾛﾎﾞｯﾄ ﾁｬｯｸ 閉端PL
Y1422  ; ﾛﾎﾞｯﾄ ﾁｬｯｸ 反転 戻し端PL
Y1423  ; ﾛﾎﾞｯﾄ ﾁｬｯｸ 反転端PL
Y1424  ; ﾛﾎﾞｯﾄ　原点復帰PL
Y1425  ; 精度確認PL
Y1430  ; 緩め部 押込み 後退端PL
Y1431  ; 緩め部 押込み 前進端PL
Y1432  ; 緩め部　ﾘﾌﾀｰ前  ｽﾄｯﾊﾟｰ　抜き端PL
Y1433  ; 緩め部　ﾘﾌﾀｰ前  ｽﾄｯﾊﾟｰ　入り端PL
Y1434  ; 穴検出部ｽﾄｯﾊﾟｰ　抜き端PL
Y1435  ; 穴検出部ｽﾄｯﾊﾟｰ　入り端PL
Y1436  ; 緩め部　NRｽﾄｯﾊﾟ-抜き端PL
Y1437  ; 緩め部　NRｽﾄｯﾊﾟ-入り端PL
Y1438  ; 緩め部　NR 位置決め 抜き端PL
Y1439  ; 緩め部　NR 位置決め 入り端PL
Y143C  ; 穴検出部位置決め抜き端PL
Y143D  ; 穴検出部位置決め入り端PL
Y143E  ; 緩め部  穴加工確認 上昇端PL
Y143F  ; 緩め部  穴加工確認 下降端PL
Y1446  ; 緩め側　搬送ﾓｰﾀｰPL
Y1450  ; 緩め部　ﾒｲﾝ NR  下降端PL
Y1451  ; 緩め部　ﾒｲﾝ NR  上昇端PL
Y1452  ; 緩め部　ﾒｲﾝ NR  起動PL
Y1453  ; 緩め部　ｻﾌﾞ NR  下降端PL
Y1454  ; 緩め部　ｻﾌﾞ NR  上昇端PL
Y1455  ; 緩め部　ｻﾌﾞ NR  起動PL
Y1460  ; 緩め側　ﾘﾌﾀｰ部　下降端PL
Y1461  ; 緩め側　ﾘﾌﾀｰ部　上昇端
Y1462  ; 緩め側　ﾘﾌﾄﾓｰﾀｰ 逆転PL
Y1463  ; 緩め側　ﾘﾌﾄﾓｰﾀｰ 正転
Y1470  ; 緩め部　ﾘﾀｰﾝｴｽｹｰﾌﾟ 後退端PL
Y1471  ; 緩め部　ﾘﾀｰﾝｴｽｹｰﾌﾟ 前進端PL
Y1472  ; ｴｱｰﾌﾞﾛｰ ｽﾄｯﾊﾟｰ  抜き端PL
Y1473  ; ｴｱｰﾌﾞﾛｰ ｽﾄｯﾊﾟｰ  入り端PL
Y1474  ; 緩め部　ｴｱｰﾌﾞﾛｰ前ｽﾄｯﾊﾟｰ抜き端PL
Y1475  ; 緩め部　ｴｱｰﾌﾞﾛｰ前ｽﾄｯﾊﾟｰ入り端PL
Y1476  ; 緩め側　ﾘﾀｰﾝCV　起動PL
Y1477  ; ｴｱｰﾌﾞﾛｰ ONPL
Y1478  ; 緩め部　ｼｬｯﾀｰ　　閉端PL
Y1479  ; 緩め部　ｼｬｯﾀｰ　　開端PL
Y147A  ; 緩めﾘﾀｰﾝCV押出前ｽﾄｯﾊﾟｰ抜き端PL
Y147B  ; 緩めﾘﾀｰﾝCV押出前ｽﾄｯﾊﾟｰ入り端PL
Y147C  ; 緩め部　ﾘﾀｰﾝCV押出ﾌﾟｯｼｬｰ後退端PL
Y147D  ; 緩め部　ﾘﾀｰﾝCV押出ﾌﾟｯｼｬｰ前進端PL
Y147E  ; 緩め部　ﾘﾀｰﾝCV押出ﾘﾌﾀｰ下降端PL
Y147F  ; 緩め部　ﾘﾀｰﾝCV押出ﾘﾌﾀｰ上昇端PL
Y1480  ; 締め部　ﾘﾌﾀｰ後　ｽﾄｯﾊﾟｰ　抜き端PL
Y1481  ; 締め部　ﾘﾌﾀｰ後　ｽﾄｯﾊﾟｰ　入り端PL
Y1482  ; 締め部　NRｽﾄｯﾊﾟｰ抜き端
Y1483  ; PL締め部　NRｽﾄｯﾊﾟｰ入り端PL
Y1484  ; 締め部　位置決め 抜き端PL
Y1485  ; 締め部　位置決め 入り端PL
Y1486  ; 締め部　ﾜｰｸ押え 戻し端PL
Y1487  ; 締め部　ﾜｰｸ押え 押え端PL
Y148A  ; 締め部　押出ｽﾄｯﾊﾟｰ 抜き端PL
Y148B  ; 締め部　押出ｽﾄｯﾊﾟｰ 入り端PL
Y148C  ; 締め部　押込み　後退端PL
Y148D  ; 締め部　押込み　前進端PL
Y148E  ; 締め部　着座確認後退端PL
Y148F  ; 締め部　着座確認前進端PL
Y1490  ; 締め部　着座確認SOL PL
Y14A0  ; 締め部　ﾅｯﾄﾗﾝﾅｰ 下降端PL
Y14A1  ; 締め部　ﾅｯﾄﾗﾝﾅｰ 上昇端PL
Y14A2  ; 締め部　ﾅｯﾄﾗﾝﾅｰ　逆転PL
Y14A3  ; 締め部　ﾅｯﾄﾗﾝﾅｰ　正転PL
Y14A4  ; 締め側　搬送ﾓｰﾀｰPL
Y14B0  ; 締め部　ﾘﾌﾀｰ 下降端PL
Y14B1  ; 締め部　ﾘﾌﾀｰ 上昇端PL
Y14B2  ; 締め側　ﾘﾌﾄﾓｰﾀｰ 逆転PL
Y14B3  ; 締め側　ﾘﾌﾄﾓｰﾀｰ 正転PL
Y14C0  ; 締め部　ﾘﾀｰﾝｴｽｹｰﾌﾟ 後退端PL
Y14C1  ; 締め部　ﾘﾀｰﾝｴｽｹｰﾌﾟ 前進端PL
Y14C2  ; 締め部　ﾘﾀｰﾝｽﾄｯﾊﾟｰ 抜き端PL
Y14C3  ; 締め部　ﾘﾀｰﾝｽﾄｯﾊﾟｰ 入り端PL
Y14C4  ; 締め側　ﾘﾀｰﾝｺﾝﾍﾞｱ 起動PL
Y14D0  ; NGﾘﾌﾀｰ　下降端PL
Y14D1  ; NGﾘﾌﾀｰ　上昇端PL
Y14E0  ; 画面　　ID1読出しPL
Y14E1  ; 画面　　ID1書込みPL
Y14E2  ; 画面　　ID2読出しPL
Y14E3  ; 画面　　ID2書込みPL
Y14E4  ; 緩め部　IDｾﾝｻｰ1 後退端PL
Y14E5  ; 緩め部　IDｾﾝｻｰ1 前進端PL
Y14E6  ; 締め部　IDｾﾝｻｰ2 後退端PL
Y14E7  ; 締め部　IDｾﾝｻｰ2 前進端PL
Y14EF  ; 画面　　ID異常PL
Y1500  ; カウント表示
Y1501  ; 気圧
Y1502  ; 運転準備
Y1503  ; 各個
Y1504  ; 連続
Y1505  ; 教示
Y1506  ; 原位置
Y1507  ; ｻｲｸﾙ中
Y150A  ; ｻｰﾎﾞON
Y150B  ; ﾌﾟﾗｸﾞOK
Y150C  ; 教示可
Y1510  ; 品番設定可
B1  ; PC電池異常
B2  ; ﾛﾎﾞｯﾄ電池異常
B3  ; ﾌﾟﾗｸﾞ異常
B4  ; ｴｱｰ圧低下
B5  ; CC-LINK異常
B6  ; ﾛﾎﾞｯﾄ異常
B7  ; ﾛﾎﾞｯﾄﾁｬｯｸ LS異常
B8  ; ﾛﾎﾞｯﾄﾁｬｯｸ 反転LS異常
B0A  ; 緩め部　押込み　LS異常
B0B  ; ｴｱｰﾌﾞﾛｰ ｽﾄｯﾊﾟｰ  LS異常
B0C  ; 穴検出部ｽﾄｯﾊﾟｰ　LS異常
B0D  ; 緩め部　NRｽﾄｯﾊﾟ-LS異常
B0E  ; 緩め部　位置決め LS異常
B0F  ; 緩め部　ﾜｰｸ押え  LS異常
B10  ; 穴検出部位置決めLS異常
B11  ; 緩め部　ﾅｯﾄﾗﾝﾅ　LS異常
B13  ; 緩め部　ﾘﾌﾀｰ LS異常
B14  ; 緩め部　ﾘﾀｰﾝｴｽｹｰﾌﾟ LS異常
B15  ; 緩め部　ｴｱｰﾌﾞﾛｰ前ｽﾄｯﾊﾟｰ　LS異常
B16  ; 緩め部　穴加工確認LS異常
B17  ; 緩め部　ｼｬｯﾀｰ　　LS異常
B18  ; 緩め部　ﾘﾌﾀｰ前  ｽﾄｯﾊﾟｰ　LS異常
B19  ; 分配部　ｼﾌﾄ LS異常
B1A  ; 分配部 着脱ﾌﾟｯｼｬｰ LS異常
B1B  ; 緩め部　ﾘﾀｰﾝCV　押出ﾌﾟｯｼｬｰLS異常
B1C  ; 緩め部 ﾘﾀｰﾝCV押出前ｽﾄｯﾊﾟｰLS異常
B1E  ; 締め部　ﾘﾀｰﾝｴｽｹｰﾌﾟ LS異常
B1F  ; 締め部 ﾘﾀｰﾝｽﾄｯﾊﾟｰ LS異常
B21  ; 予備
B22  ; 締め部　ﾘﾌﾀｰ LS異常
B23  ; 締め部　ﾘﾌﾀｰ後　ｽﾄｯﾊﾟｰ　LS異常
B24  ; 締め部　NRｽﾄｯﾊﾟｰLS異常
B25  ; 締め部　位置決め LS異常
B26  ; 締め部 ﾊﾟﾚｯﾄ押え LS異常
B28  ; 締め部　押出ｽﾄｯﾊﾟｰ LS異常
B29  ; 締め部　押込み　LS異常
B2A  ; 締め部 ﾅｯﾄﾗﾝﾅｰ　LS異常
B2B  ; 締め部　着座確認LS異常
B2C  ; NGﾘﾌﾀｰ　LS異常
B2D  ; 締め部　IDｾﾝｻｰ　LS異常
B30  ; 穴検出　NG
B31  ; 穴検出　治具折れ異常
B32  ; 緩め部　ｴｱｰﾓｰﾀｰ ﾎﾞﾙﾄ緩め異常
B37  ; 締め部　ﾅｯﾄﾗﾝﾅｼｽﾃﾑ異常
B38  ; 締め部　ﾅｯﾄﾗﾝﾅ締付 NG(ﾄﾙｸ)
B39  ; 締め部　ﾅｯﾄﾗﾝﾅ締付NG(角度)
B3C  ; NGｼｭｰﾄ　満載
B41  ; ﾊﾟﾚｯﾄID異常
B42  ; ID1読み出し異常
B44  ; ID2読み出し異常
B46  ; ID異常
B47  ; 緩め側搬送CV INV異常
B48  ; 緩め側ﾘﾌﾄﾓｰﾀｰ ｻｰﾏﾙﾄﾘｯﾌﾟ
B49  ; 緩め側ﾘﾀｰﾝCV INV異常
B4A  ; 締め側搬送CV INV異常
B4B  ; 締め側ﾘﾌﾄﾓｰﾀｰ ｻｰﾏﾙﾄﾘｯﾌﾟ
B4C  ; 締め側ﾘﾀｰﾝCV INV異常
B4F  ; ﾛﾎﾞｯﾄﾁｬｯｸ動作異常
B50  ; 緩め部　押込み 動作異常
B51  ; ｴｱｰﾌﾞﾛｰ ｽﾄｯﾊﾟｰ　動作異常
B52  ; 穴検出部ｽﾄｯﾊﾟｰ　動作異常
B53  ; 緩め部　NRｽﾄｯﾊﾟ-動作異常
B54  ; 緩め部　位置決め動作異常
B56  ; 穴検出部位置決め動作異常
B57  ; 緩め部　ﾅｯﾄﾗﾝﾅｰ 動作異常
B59  ; 緩め部　ﾘﾌﾀｰ 動作異常
B5A  ; 緩め部　ﾘﾀｰﾝｴｽｹｰﾌﾟ 動作異常
B5B  ; 緩め部　ｴｱｰﾌﾞﾛｰ前ｽﾄｯﾊﾟｰ動作異常
B5C  ; 緩め部 穴加工確認動作異常
B5D  ; 緩め部　ｼｬｯﾀｰ　　動作異常
B5E  ; 緩め部　ﾘﾌﾀｰ前  ｽﾄｯﾊﾟｰ　動作異常
B61  ; 緩め部　ﾘﾀｰﾝCV押出ﾌﾟｯｼｬｰ動作異常
B62  ; 緩め部ﾘﾀｰﾝCV押出前ｽﾄｯﾊﾟｰ動作異常
B63  ; 分配部　ｼﾌﾄ 動作異常
B64  ; 分配部　着脱ﾌﾟｯｼｬｰ 動作異常
B65  ; 着座つまり検知
B66  ; 締め部　ﾘﾀｰﾝｴｽｹｰﾌﾟ 動作異常
B67  ; 締め部　ﾘﾀｰﾝｽﾄｯﾊﾟｰ 動作異常
B68  ; 締め部 ﾘﾌﾀｰ 動作異常
B69  ; 締め部　着座確認　動作異常
B6A  ; NGﾘﾌﾀｰ　動作異常
B6B  ; 締め部　IDｾﾝｻｰ　動作異常
B6C  ; 締め部　ﾘﾌﾀｰ後　ｽﾄｯﾊﾟｰ　動作異常
B6D  ; 締め部　NRｽﾄｯﾊﾟｰ動作異常
B6E  ; 締め部　位置決め 動作異常
B6F  ; 締め部　ﾊﾟﾚｯﾄ押え 動作異常
B70  ; 締め部　押出ｽﾄｯﾊﾟｰ 動作異常
B71  ; 締め部　押込み　動作異常
B72  ; 締め部　ﾅｯﾄﾗﾝﾅｰ 動作異常
B73  ; 緩め部　ﾅｯﾄﾗﾝﾅ　ﾀｲﾑｵｰﾊﾞｰ
B7A  ; 分配部⇒緩め側　押込み　流動異常
B7B  ; 穴検出部ﾊﾟﾚｯﾄ排出流動異常
B7C  ; 緩めNR⇒ﾘﾌﾀ ﾊﾟﾚｯﾄ排出流動異常
B7D  ; 緩め部ﾘﾌﾀ⇒ﾘﾀｰﾝ ﾊﾟﾚｯﾄ流動異常
B7E  ; ｴｱｰﾌﾞﾛｰ ﾊﾟﾚｯﾄ排出流動異常
B7F  ; 締め部　ﾘﾀｰﾝ⇒ﾘﾌﾀ ﾊﾟﾚｯﾄ流動異常
B80  ; 締め部　ﾘﾌﾀｰ ﾊﾟﾚｯﾄ流動異常
B81  ; 締め部　ﾅｯﾄﾗﾝﾅｰ部 ﾊﾟﾚｯﾄ流動異常
B82  ; 締め側CV⇒分配部 ﾊﾟﾚｯﾄ流動異常
B86  ; ﾊﾟﾚｯﾄ着座異常
D8  ; 画面切替
D7000  ; 品番検索結果
D7001  ; 品番一致数
D7002  ; 品番検索結果*2
T1  ; 電源入り確認2
T12  ; 着座無効
T13  ; 着座有効
T16  ; 教示モード
T20  ; ｴｱｰ元圧低下
T21  ; ﾛﾎﾞｯﾄﾁｬｯｸ動作異常
T30  ; 緩め部　押込み　動作異常
T31  ; ｴｱｰﾌﾞﾛｰ ｽﾄｯﾊﾟｰ　動作異常
T32  ; 穴検出部ｽﾄｯﾊﾟｰ　動作異常
T33  ; 緩め部　NRｽﾄｯﾊﾟ-動作異常
T34  ; 緩め部　位置決め動作異常
T36  ; 穴検出部位置決め動作異常
T37  ; 緩め部　ﾅｯﾄﾗﾝﾅｰ 動作異常
T39  ; 緩め部　ﾘﾌﾀｰ 動作異常
T40  ; 緩め部　ﾘﾀｰﾝｴｽｹｰﾌﾟ 動作異常
T41  ; 緩め部　ｴｱｰﾌﾞﾛｰ前ｽﾄｯﾊﾟｰ動作異常
T42  ; 緩め部 穴加工確認動作異常
T43  ; 緩め部　ｼｬｯﾀｰ　　動作異常
T44  ; 緩め部　ﾘﾌﾀｰ前  ｽﾄｯﾊﾟｰ　動作異常
T47  ; 緩め部　ﾘﾀｰﾝCV押出ﾌﾟｯｼｬｰ動作異常
T48  ; 緩め部ﾘﾀｰﾝCV押出前ｽﾄｯﾊﾟｰ動作異常
T50  ; 分配部　ｼﾌﾄ 動作異常
T51  ; 分配部　着脱ﾌﾟｯｼｬｰ 動作異常
T55  ; ﾊﾟﾚｯﾄ着座異常
T57  ; 着座つまり検知
T60  ; 締め部　ﾘﾀｰﾝｴｽｹｰﾌﾟ 動作異常
T61  ; 締め部　ﾘﾀｰﾝｽﾄｯﾊﾟｰ 動作異常
T62  ; 締め部 ﾘﾌﾀｰ 動作異常
T63  ; 締め部　着座確認　動作異常
T64  ; NGﾘﾌﾀｰ　動作異常
T65  ; 締め部　IDｾﾝｻｰ　動作異常
T66  ; 締め部　ﾘﾌﾀｰ後　ｽﾄｯﾊﾟｰ　動作異常
T67  ; 締め部　NRｽﾄｯﾊﾟｰ動作異常
T68  ; 締め部　位置決め 動作異常
T71  ; 締め部　押出ｽﾄｯﾊﾟｰ 動作異常
T72  ; 締め部　押込み　動作異常
T73  ; 締め部　ﾅｯﾄﾗﾝﾅｰ 動作異常
T90  ; 分配部⇒緩め側　押込み　流動異常
T91  ; 穴検出部ﾊﾟﾚｯﾄ排出流動異常
T92  ; 緩めNR⇒ﾘﾌﾀ ﾊﾟﾚｯﾄ排出流動異常
T93  ; 緩め部ﾘﾌﾀ⇒ﾘﾀｰﾝ ﾊﾟﾚｯﾄ流動異常
T94  ; ｴｱｰﾌﾞﾛｰ ﾊﾟﾚｯﾄ排出流動異常
T95  ; 締め部　ﾘﾀｰﾝ⇒ﾘﾌﾀ ﾊﾟﾚｯﾄ流動異常
T96  ; 締め部　ﾘﾌﾀｰ ﾊﾟﾚｯﾄ流動異常
T97  ; 締め部　ﾅｯﾄﾗﾝﾅｰ部 ﾊﾟﾚｯﾄ流動異常
T98  ; 締め側CV⇒分配部 ﾊﾟﾚｯﾄ流動異常
T100  ; ﾛﾎﾞｯﾄﾁｬｯｸ開端OFF
T106  ; ID1読出しﾀｲﾑｵｰﾊﾞｰ
T107  ; ID1書込みﾀｲﾑｵｰﾊﾞｰ
T108  ; ID2読出しﾀｲﾑｵｰﾊﾞｰ
T109  ; ID2書込みﾀｲﾑｵｰﾊﾞｰ
T116  ; ﾅｯﾄﾗﾝﾅ　出力切替終了
T117  ; ﾅｯﾄﾗﾝﾅ　BANK 0
T118  ; ﾅｯﾄﾗﾝﾅ　BANK 2
T140  ; ｴｱｰﾌﾞﾛｰ ON時間
T141  ; ｴｱｰﾌﾞﾛｰ OFF時間
T250  ; ID1　 　読出し　TRG
T254  ; ID1 読出し完了
T259  ; カウント表示時間
T264  ; ID2 読出し完了
T307  ; 緩め部　NR 位置決抜き端　ﾀｲﾏ
T309  ; 穴検出部ｽﾄｯﾊﾟｰ　抜き端　ﾀｲﾏ
T313  ; 緩め部  穴検出　上昇端
T315  ; 緩め部　ﾒｲﾝ NR  上昇端　ﾀｲﾏ
T317  ; 緩め部　IDｾﾝｻｰ　前進端ﾀｲﾏ
T318  ; 緩め部　IDｾﾝｻｰ　後退端ﾀｲﾏ
T321  ; 緩め部　ｻﾌﾞ NR  下降端　ﾀｲﾏ
T331  ; 緩め部 ﾘﾀｰﾝCV押出前ｽﾄｯﾊﾟｰ抜き端
T334  ; 緩め部　ﾘﾀｰﾝCV　押出ﾌﾟｯｼｬｰ前進端
T341  ; 締め部　ﾘﾀｰﾝｽﾄｯﾊﾟｰ 抜き端ﾀｲﾏ
T342  ; 締め部　ﾘﾌﾀｰ 　　上昇端　ﾀｲﾏ
T343  ; 締め部　ﾘﾌﾀｰ 　　下降端　ﾀｲﾏ
T350  ; 締め部　IDｾﾝｻｰ　前進端ﾀｲﾏ
T351  ; 締め部　IDｾﾝｻｰ　後退端ﾀｲﾏ
T352  ; 締め部　ﾜｰｸ押え 押え端ﾀｲﾏ
T353  ; 締め部　ﾜｰｸ押え 戻し端ﾀｲﾏ
T354  ; 締め部　着座確認前進端ﾀｲﾏ
T355  ; 締め部　着座確認後退端ﾀｲﾏ
T666  ; ID1 TRG ON確認 ﾀｲﾏ
T777  ; ID2 TRG ON確認ﾀｲﾏ
